KUKA KRL program: unicorn2_1.src

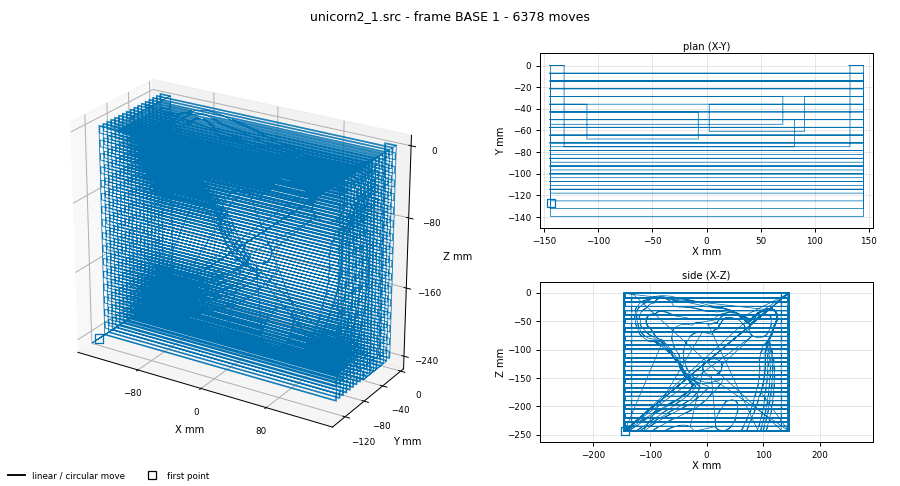
[picture p0: tool path of unicorn2_1.src in frame BASE 1, 6378 of 6379 moves have a stored position in this frame; points joined in program order, loops and branches not executed]
&ACCESS RVP
&REL 1
&PARAM TEMPLATE = C:\KRC\Roboter\Template\vorgabe
&PARAM EDITMASK = *
DEF unicorn2_1( )
EXT BAS (BAS_COMMAND :IN,REAL :IN )

INT INDX
FOR INDX=1 TO 6
	$ACC_AXIS[INDX]=50
	$VEL_AXIS[INDX]=20
ENDFOR

$VEL.ORI1=200
$VEL.ORI2=200
$ACC.ORI1=100
$ACC.ORI2=100

$VEL.CP = 0.2
$ACC.CP = 5

$IPO_MODE = #BASE
$APO.CDIS = 0.5
$ADVANCE = 5

$ACT_TOOL = 1
$TOOL=TOOL_DATA[1]
$ACT_BASE = 1
$BASE=BASE_DATA[1]

PTP {A1 30.0,A2 -90.0,A3 90.0,A4 0.0,A5 90.0,A6 0.0}

LIN {X -144.015,Y -126.800,Z -242.561,A -90.000,B 90.000,C 0.000} C_DIS
LIN {X -144.015,Y -114.300,Z -242.561,A -90.000,B 90.000,C 0.000} C_DIS
LIN {X 144.015,Y -114.300,Z -242.561,A -90.000,B 90.000,C 0.000} C_DIS
LIN {X 144.015,Y -114.300,Z -235.012,A -90.000,B 90.000,C 0.000} C_DIS
LIN {X -144.015,Y -114.300,Z -235.012,A -90.000,B 90.000,C 0.000} C_DIS
LIN {X -144.015,Y -114.300,Z -227.464,A -90.000,B 90.000,C 0.000} C_DIS
LIN {X 144.015,Y -114.300,Z -227.464,A -90.000,B 90.000,C 0.000} C_DIS
LIN {X 144.015,Y -114.300,Z -219.915,A -90.000,B 90.000,C 0.000} C_DIS
LIN {X -144.015,Y -114.300,Z -219.915,A -90.000,B 90.000,C 0.000} C_DIS
LIN {X -144.015,Y -114.300,Z -212.366,A -90.000,B 90.000,C 0.000} C_DIS
LIN {X 144.015,Y -114.300,Z -212.366,A -90.000,B 90.000,C 0.000} C_DIS
LIN {X 144.015,Y -114.300,Z -204.817,A -90.000,B 90.000,C 0.000} C_DIS
LIN {X -144.015,Y -114.300,Z -204.817,A -90.000,B 90.000,C 0.000} C_DIS
LIN {X -144.015,Y -114.300,Z -197.269,A -90.000,B 90.000,C 0.000} C_DIS
LIN {X 144.015,Y -114.300,Z -197.269,A -90.000,B 90.000,C 0.000} C_DIS
LIN {X 144.015,Y -114.300,Z -189.720,A -90.000,B 90.000,C 0.000} C_DIS
LIN {X -144.015,Y -114.300,Z -189.720,A -90.000,B 90.000,C 0.000} C_DIS
LIN {X -144.015,Y -114.300,Z -182.171,A -90.000,B 90.000,C 0.000} C_DIS
LIN {X 144.015,Y -114.300,Z -182.171,A -90.000,B 90.000,C 0.000} C_DIS
LIN {X 144.015,Y -114.300,Z -174.622,A -90.000,B 90.000,C 0.000} C_DIS
LIN {X -144.015,Y -114.300,Z -174.622,A -90.000,B 90.000,C 0.000} C_DIS
LIN {X -144.015,Y -114.300,Z -167.073,A -90.000,B 90.000,C 0.000} C_DIS
LIN {X 144.015,Y -114.300,Z -167.073,A -90.000,B 90.000,C 0.000} C_DIS
LIN {X 144.015,Y -114.300,Z -159.525,A -90.000,B 90.000,C 0.000} C_DIS
LIN {X -144.015,Y -114.300,Z -159.525,A -90.000,B 90.000,C 0.000} C_DIS
LIN {X -144.015,Y -114.300,Z -151.976,A -90.000,B 90.000,C 0.000} C_DIS
LIN {X 144.015,Y -114.300,Z -151.976,A -90.000,B 90.000,C 0.000} C_DIS
LIN {X 144.015,Y -114.300,Z -144.427,A -90.000,B 90.000,C 0.000} C_DIS
LIN {X -144.015,Y -114.300,Z -144.427,A -90.000,B 90.000,C 0.000} C_DIS
LIN {X -144.015,Y -114.300,Z -136.878,A -90.000,B 90.000,C 0.000} C_DIS
LIN {X 144.015,Y -114.300,Z -136.878,A -90.000,B 90.000,C 0.000} C_DIS
LIN {X 144.015,Y -114.300,Z -129.329,A -90.000,B 90.000,C 0.000} C_DIS
LIN {X -144.015,Y -114.300,Z -129.329,A -90.000,B 90.000,C 0.000} C_DIS
LIN {X -144.015,Y -114.300,Z -121.781,A -90.000,B 90.000,C 0.000} C_DIS
LIN {X 144.015,Y -114.300,Z -121.781,A -90.000,B 90.000,C 0.000} C_DIS
LIN {X 144.015,Y -114.300,Z -114.232,A -90.000,B 90.000,C 0.000} C_DIS
LIN {X -144.015,Y -114.300,Z -114.232,A -90.000,B 90.000,C 0.000} C_DIS
LIN {X -144.015,Y -114.300,Z -106.683,A -90.000,B 90.000,C 0.000} C_DIS
LIN {X 144.015,Y -114.300,Z -106.683,A -90.000,B 90.000,C 0.000} C_DIS
LIN {X 144.015,Y -114.300,Z -99.134,A -90.000,B 90.000,C 0.000} C_DIS
LIN {X -144.015,Y -114.300,Z -99.134,A -90.000,B 90.000,C 0.000} C_DIS
LIN {X -144.015,Y -114.300,Z -91.586,A -90.000,B 90.000,C 0.000} C_DIS
LIN {X 144.015,Y -114.300,Z -91.586,A -90.000,B 90.000,C 0.000} C_DIS
LIN {X 144.015,Y -114.300,Z -84.037,A -90.000,B 90.000,C 0.000} C_DIS
LIN {X -144.015,Y -114.300,Z -84.037,A -90.000,B 90.000,C 0.000} C_DIS
LIN {X -144.015,Y -114.300,Z -76.488,A -90.000,B 90.000,C 0.000} C_DIS
LIN {X 144.015,Y -114.300,Z -76.488,A -90.000,B 90.000,C 0.000} C_DIS
LIN {X 144.015,Y -114.300,Z -68.939,A -90.000,B 90.000,C 0.000} C_DIS
LIN {X -144.015,Y -114.300,Z -68.939,A -90.000,B 90.000,C 0.000} C_DIS
LIN {X -144.015,Y -114.300,Z -61.390,A -90.000,B 90.000,C 0.000} C_DIS
LIN {X 144.015,Y -114.300,Z -61.390,A -90.000,B 90.000,C 0.000} C_DIS
LIN {X 144.015,Y -114.300,Z -53.842,A -90.000,B 90.000,C 0.000} C_DIS
LIN {X -144.015,Y -114.300,Z -53.842,A -90.000,B 90.000,C 0.000} C_DIS
LIN {X -144.015,Y -114.300,Z -46.293,A -90.000,B 90.000,C 0.000} C_DIS
LIN {X 144.015,Y -114.300,Z -46.293,A -90.000,B 90.000,C 0.000} C_DIS
LIN {X 144.015,Y -114.300,Z -38.744,A -90.000,B 90.000,C 0.000} C_DIS
LIN {X -144.015,Y -114.300,Z -38.744,A -90.000,B 90.000,C 0.000} C_DIS
LIN {X -144.015,Y -114.300,Z -31.195,A -90.000,B 90.000,C 0.000} C_DIS
LIN {X 144.015,Y -114.300,Z -31.195,A -90.000,B 90.000,C 0.000} C_DIS
LIN {X 144.015,Y -114.300,Z -23.646,A -90.000,B 90.000,C 0.000} C_DIS
LIN {X -144.015,Y -114.300,Z -23.646,A -90.000,B 90.000,C 0.000} C_DIS
LIN {X -144.015,Y -114.300,Z -16.098,A -90.000,B 90.000,C 0.000} C_DIS
LIN {X 144.015,Y -114.300,Z -16.098,A -90.000,B 90.000,C 0.000} C_DIS
LIN {X 144.015,Y -114.300,Z -8.549,A -90.000,B 90.000,C 0.000} C_DIS
LIN {X -144.015,Y -114.300,Z -8.549,A -90.000,B 90.000,C 0.000} C_DIS
LIN {X -144.015,Y -114.300,Z -1.000,A -90.000,B 90.000,C 0.000} C_DIS
LIN {X 144.015,Y -114.300,Z -1.000,A -90.000,B 90.000,C 0.000} C_DIS
LIN {X 145.015,Y -114.300,Z 0.000,A -90.000,B 90.000,C 0.000} C_DIS
LIN {X -145.015,Y -114.300,Z 0.000,A -90.000,B 90.000,C 0.000} C_DIS
LIN {X -145.015,Y -114.300,Z -243.561,A -90.000,B 90.000,C 0.000} C_DIS
LIN {X 145.015,Y -114.300,Z -243.561,A -90.000,B 90.000,C 0.000} C_DIS
LIN {X 145.015,Y -114.300,Z 0.000,A -90.000,B 90.000,C 0.000} C_DIS
LIN {X 145.015,Y -126.800,Z 0.000,A -90.000,B 90.000,C 0.000} C_DIS
LIN {X 145.015,Y -139.300,Z 0.000,A -90.000,B 90.000,C 0.000} C_DIS
LIN {X -144.015,Y -139.300,Z -242.561,A -90.000,B 90.000,C 0.000} C_DIS
LIN {X -144.015,Y -132.156,Z -242.561,A -90.000,B 90.000,C 0.000} C_DIS
LIN {X -144.015,Y -119.656,Z -242.561,A -90.000,B 90.000,C 0.000} C_DIS
LIN {X -144.015,Y -107.156,Z -242.561,A -90.000,B 90.000,C 0.000} C_DIS
LIN {X 144.015,Y -107.156,Z -242.561,A -90.000,B 90.000,C 0.000} C_DIS
LIN {X 144.015,Y -107.156,Z -235.012,A -90.000,B 90.000,C 0.000} C_DIS
LIN {X -144.015,Y -107.156,Z -235.012,A -90.000,B 90.000,C 0.000} C_DIS
LIN {X -144.015,Y -107.156,Z -227.464,A -90.000,B 90.000,C 0.000} C_DIS
LIN {X 144.015,Y -107.156,Z -227.464,A -90.000,B 90.000,C 0.000} C_DIS
LIN {X 144.015,Y -107.156,Z -219.915,A -90.000,B 90.000,C 0.000} C_DIS
LIN {X -144.015,Y -107.156,Z -219.915,A -90.000,B 90.000,C 0.000} C_DIS
LIN {X -144.015,Y -107.156,Z -212.366,A -90.000,B 90.000,C 0.000} C_DIS
LIN {X 144.015,Y -107.156,Z -212.366,A -90.000,B 90.000,C 0.000} C_DIS
LIN {X 144.015,Y -107.156,Z -204.817,A -90.000,B 90.000,C 0.000} C_DIS
LIN {X -144.015,Y -107.156,Z -204.817,A -90.000,B 90.000,C 0.000} C_DIS
LIN {X -144.015,Y -107.156,Z -197.269,A -90.000,B 90.000,C 0.000} C_DIS
LIN {X 144.015,Y -107.156,Z -197.269,A -90.000,B 90.000,C 0.000} C_DIS
LIN {X 144.015,Y -107.156,Z -189.720,A -90.000,B 90.000,C 0.000} C_DIS
LIN {X -144.015,Y -107.156,Z -189.720,A -90.000,B 90.000,C 0.000} C_DIS
LIN {X -144.015,Y -107.156,Z -182.171,A -90.000,B 90.000,C 0.000} C_DIS
LIN {X 144.015,Y -107.156,Z -182.171,A -90.000,B 90.000,C 0.000} C_DIS
LIN {X 144.015,Y -107.156,Z -174.622,A -90.000,B 90.000,C 0.000} C_DIS
LIN {X -144.015,Y -107.156,Z -174.622,A -90.000,B 90.000,C 0.000} C_DIS
LIN {X -144.015,Y -107.156,Z -167.073,A -90.000,B 90.000,C 0.000} C_DIS
LIN {X 144.015,Y -107.156,Z -167.073,A -90.000,B 90.000,C 0.000} C_DIS
LIN {X 144.015,Y -107.156,Z -159.525,A -90.000,B 90.000,C 0.000} C_DIS
LIN {X -144.015,Y -107.156,Z -159.525,A -90.000,B 90.000,C 0.000} C_DIS
LIN {X -144.015,Y -107.156,Z -151.976,A -90.000,B 90.000,C 0.000} C_DIS
LIN {X 144.015,Y -107.156,Z -151.976,A -90.000,B 90.000,C 0.000} C_DIS
LIN {X 144.015,Y -107.156,Z -144.427,A -90.000,B 90.000,C 0.000} C_DIS
LIN {X -144.015,Y -107.156,Z -144.427,A -90.000,B 90.000,C 0.000} C_DIS
LIN {X -144.015,Y -107.156,Z -136.878,A -90.000,B 90.000,C 0.000} C_DIS
LIN {X 144.015,Y -107.156,Z -136.878,A -90.000,B 90.000,C 0.000} C_DIS
LIN {X 144.015,Y -107.156,Z -129.329,A -90.000,B 90.000,C 0.000} C_DIS
LIN {X -144.015,Y -107.156,Z -129.329,A -90.000,B 90.000,C 0.000} C_DIS
LIN {X -144.015,Y -107.156,Z -121.781,A -90.000,B 90.000,C 0.000} C_DIS
LIN {X 144.015,Y -107.156,Z -121.781,A -90.000,B 90.000,C 0.000} C_DIS
LIN {X 144.015,Y -107.156,Z -114.232,A -90.000,B 90.000,C 0.000} C_DIS
LIN {X -144.015,Y -107.156,Z -114.232,A -90.000,B 90.000,C 0.000} C_DIS
LIN {X -144.015,Y -107.156,Z -106.683,A -90.000,B 90.000,C 0.000} C_DIS
LIN {X 144.015,Y -107.156,Z -106.683,A -90.000,B 90.000,C 0.000} C_DIS
LIN {X 144.015,Y -107.156,Z -99.134,A -90.000,B 90.000,C 0.000} C_DIS
LIN {X -144.015,Y -107.156,Z -99.134,A -90.000,B 90.000,C 0.000} C_DIS
LIN {X -144.015,Y -107.156,Z -91.586,A -90.000,B 90.000,C 0.000} C_DIS
LIN {X 144.015,Y -107.156,Z -91.586,A -90.000,B 90.000,C 0.000} C_DIS
LIN {X 144.015,Y -107.156,Z -84.037,A -90.000,B 90.000,C 0.000} C_DIS
LIN {X -144.015,Y -107.156,Z -84.037,A -90.000,B 90.000,C 0.000} C_DIS
LIN {X -144.015,Y -107.156,Z -76.488,A -90.000,B 90.000,C 0.000} C_DIS
LIN {X 144.015,Y -107.156,Z -76.488,A -90.000,B 90.000,C 0.000} C_DIS
LIN {X 144.015,Y -107.156,Z -68.939,A -90.000,B 90.000,C 0.000} C_DIS
LIN {X -144.015,Y -107.156,Z -68.939,A -90.000,B 90.000,C 0.000} C_DIS
LIN {X -144.015,Y -107.156,Z -61.390,A -90.000,B 90.000,C 0.000} C_DIS
LIN {X 144.015,Y -107.156,Z -61.390,A -90.000,B 90.000,C 0.000} C_DIS
LIN {X 144.015,Y -107.156,Z -53.842,A -90.000,B 90.000,C 0.000} C_DIS
LIN {X -144.015,Y -107.156,Z -53.842,A -90.000,B 90.000,C 0.000} C_DIS
LIN {X -144.015,Y -107.156,Z -46.293,A -90.000,B 90.000,C 0.000} C_DIS
LIN {X 144.015,Y -107.156,Z -46.293,A -90.000,B 90.000,C 0.000} C_DIS
LIN {X 144.015,Y -107.156,Z -38.744,A -90.000,B 90.000,C 0.000} C_DIS
LIN {X -144.015,Y -107.156,Z -38.744,A -90.000,B 90.000,C 0.000} C_DIS
LIN {X -144.015,Y -107.156,Z -31.195,A -90.000,B 90.000,C 0.000} C_DIS
LIN {X 144.015,Y -107.156,Z -31.195,A -90.000,B 90.000,C 0.000} C_DIS
LIN {X 144.015,Y -107.156,Z -23.646,A -90.000,B 90.000,C 0.000} C_DIS
LIN {X -144.015,Y -107.156,Z -23.646,A -90.000,B 90.000,C 0.000} C_DIS
LIN {X -144.015,Y -107.156,Z -16.098,A -90.000,B 90.000,C 0.000} C_DIS
LIN {X 144.015,Y -107.156,Z -16.098,A -90.000,B 90.000,C 0.000} C_DIS
LIN {X 144.015,Y -107.156,Z -8.549,A -90.000,B 90.000,C 0.000} C_DIS
LIN {X -144.015,Y -107.156,Z -8.549,A -90.000,B 90.000,C 0.000} C_DIS
LIN {X -144.015,Y -107.156,Z -1.000,A -90.000,B 90.000,C 0.000} C_DIS
LIN {X 144.015,Y -107.156,Z -1.000,A -90.000,B 90.000,C 0.000} C_DIS
LIN {X 145.015,Y -107.156,Z 0.000,A -90.000,B 90.000,C 0.000} C_DIS
LIN {X -145.015,Y -107.156,Z 0.000,A -90.000,B 90.000,C 0.000} C_DIS
LIN {X -145.015,Y -107.156,Z -243.561,A -90.000,B 90.000,C 0.000} C_DIS
LIN {X 145.015,Y -107.156,Z -243.561,A -90.000,B 90.000,C 0.000} C_DIS
LIN {X 145.015,Y -107.156,Z 0.000,A -90.000,B 90.000,C 0.000} C_DIS
LIN {X 145.015,Y -119.656,Z 0.000,A -90.000,B 90.000,C 0.000} C_DIS
LIN {X 145.015,Y -132.156,Z 0.000,A -90.000,B 90.000,C 0.000} C_DIS
LIN {X -144.015,Y -132.156,Z -242.561,A -90.000,B 90.000,C 0.000} C_DIS
LIN {X -144.015,Y -125.013,Z -242.561,A -90.000,B 90.000,C 0.000} C_DIS
LIN {X -144.015,Y -112.513,Z -242.561,A -90.000,B 90.000,C 0.000} C_DIS
LIN {X -144.015,Y -100.013,Z -242.561,A -90.000,B 90.000,C 0.000} C_DIS
LIN {X 144.015,Y -100.013,Z -242.561,A -90.000,B 90.000,C 0.000} C_DIS
LIN {X 144.015,Y -100.013,Z -235.012,A -90.000,B 90.000,C 0.000} C_DIS
LIN {X -144.015,Y -100.013,Z -235.012,A -90.000,B 90.000,C 0.000} C_DIS
LIN {X -144.015,Y -100.013,Z -227.464,A -90.000,B 90.000,C 0.000} C_DIS
LIN {X 144.015,Y -100.013,Z -227.464,A -90.000,B 90.000,C 0.000} C_DIS
LIN {X 144.015,Y -100.013,Z -219.915,A -90.000,B 90.000,C 0.000} C_DIS
LIN {X -144.015,Y -100.013,Z -219.915,A -90.000,B 90.000,C 0.000} C_DIS
LIN {X -144.015,Y -100.013,Z -212.366,A -90.000,B 90.000,C 0.000} C_DIS
LIN {X 144.015,Y -100.013,Z -212.366,A -90.000,B 90.000,C 0.000} C_DIS
LIN {X 144.015,Y -100.013,Z -204.817,A -90.000,B 90.000,C 0.000} C_DIS
LIN {X -144.015,Y -100.013,Z -204.817,A -90.000,B 90.000,C 0.000} C_DIS
LIN {X -144.015,Y -100.013,Z -197.269,A -90.000,B 90.000,C 0.000} C_DIS
LIN {X 144.015,Y -100.013,Z -197.269,A -90.000,B 90.000,C 0.000} C_DIS
LIN {X 144.015,Y -100.013,Z -189.720,A -90.000,B 90.000,C 0.000} C_DIS
LIN {X -144.015,Y -100.013,Z -189.720,A -90.000,B 90.000,C 0.000} C_DIS
LIN {X -144.015,Y -100.013,Z -182.171,A -90.000,B 90.000,C 0.000} C_DIS
LIN {X 144.015,Y -100.013,Z -182.171,A -90.000,B 90.000,C 0.000} C_DIS
LIN {X 144.015,Y -100.013,Z -174.622,A -90.000,B 90.000,C 0.000} C_DIS
LIN {X -144.015,Y -100.013,Z -174.622,A -90.000,B 90.000,C 0.000} C_DIS
LIN {X -144.015,Y -100.013,Z -167.073,A -90.000,B 90.000,C 0.000} C_DIS
LIN {X 144.015,Y -100.013,Z -167.073,A -90.000,B 90.000,C 0.000} C_DIS
LIN {X 144.015,Y -100.013,Z -159.525,A -90.000,B 90.000,C 0.000} C_DIS
LIN {X -144.015,Y -100.013,Z -159.525,A -90.000,B 90.000,C 0.000} C_DIS
LIN {X -144.015,Y -100.013,Z -151.976,A -90.000,B 90.000,C 0.000} C_DIS
LIN {X 144.015,Y -100.013,Z -151.976,A -90.000,B 90.000,C 0.000} C_DIS
LIN {X 144.015,Y -100.013,Z -144.427,A -90.000,B 90.000,C 0.000} C_DIS
LIN {X -144.015,Y -100.013,Z -144.427,A -90.000,B 90.000,C 0.000} C_DIS
LIN {X -144.015,Y -100.013,Z -136.878,A -90.000,B 90.000,C 0.000} C_DIS
LIN {X 144.015,Y -100.013,Z -136.878,A -90.000,B 90.000,C 0.000} C_DIS
LIN {X 144.015,Y -100.013,Z -129.329,A -90.000,B 90.000,C 0.000} C_DIS
LIN {X -144.015,Y -100.013,Z -129.329,A -90.000,B 90.000,C 0.000} C_DIS
LIN {X -144.015,Y -100.013,Z -121.781,A -90.000,B 90.000,C 0.000} C_DIS
LIN {X 144.015,Y -100.013,Z -121.781,A -90.000,B 90.000,C 0.000} C_DIS
LIN {X 144.015,Y -100.013,Z -114.232,A -90.000,B 90.000,C 0.000} C_DIS
LIN {X -144.015,Y -100.013,Z -114.232,A -90.000,B 90.000,C 0.000} C_DIS
LIN {X -144.015,Y -100.013,Z -106.683,A -90.000,B 90.000,C 0.000} C_DIS
LIN {X 144.015,Y -100.013,Z -106.683,A -90.000,B 90.000,C 0.000} C_DIS
LIN {X 144.015,Y -100.013,Z -99.134,A -90.000,B 90.000,C 0.000} C_DIS
LIN {X -144.015,Y -100.013,Z -99.134,A -90.000,B 90.000,C 0.000} C_DIS
LIN {X -144.015,Y -100.013,Z -91.586,A -90.000,B 90.000,C 0.000} C_DIS
LIN {X 144.015,Y -100.013,Z -91.586,A -90.000,B 90.000,C 0.000} C_DIS
LIN {X 144.015,Y -100.013,Z -84.037,A -90.000,B 90.000,C 0.000} C_DIS
LIN {X -144.015,Y -100.013,Z -84.037,A -90.000,B 90.000,C 0.000} C_DIS
LIN {X -144.015,Y -100.013,Z -76.488,A -90.000,B 90.000,C 0.000} C_DIS
LIN {X 144.015,Y -100.013,Z -76.488,A -90.000,B 90.000,C 0.000} C_DIS
LIN {X 144.015,Y -100.013,Z -68.939,A -90.000,B 90.000,C 0.000} C_DIS
LIN {X -144.015,Y -100.013,Z -68.939,A -90.000,B 90.000,C 0.000} C_DIS
LIN {X -144.015,Y -100.013,Z -61.390,A -90.000,B 90.000,C 0.000} C_DIS
LIN {X 144.015,Y -100.013,Z -61.390,A -90.000,B 90.000,C 0.000} C_DIS
LIN {X 144.015,Y -100.013,Z -53.842,A -90.000,B 90.000,C 0.000} C_DIS
LIN {X -144.015,Y -100.013,Z -53.842,A -90.000,B 90.000,C 0.000} C_DIS
LIN {X -144.015,Y -100.013,Z -46.293,A -90.000,B 90.000,C 0.000} C_DIS
LIN {X 144.015,Y -100.013,Z -46.293,A -90.000,B 90.000,C 0.000} C_DIS
LIN {X 144.015,Y -100.013,Z -38.744,A -90.000,B 90.000,C 0.000} C_DIS
LIN {X -144.015,Y -100.013,Z -38.744,A -90.000,B 90.000,C 0.000} C_DIS
LIN {X -144.015,Y -100.013,Z -31.195,A -90.000,B 90.000,C 0.000} C_DIS
LIN {X 144.015,Y -100.013,Z -31.195,A -90.000,B 90.000,C 0.000} C_DIS
LIN {X 144.015,Y -100.013,Z -23.646,A -90.000,B 90.000,C 0.000} C_DIS
LIN {X -144.015,Y -100.013,Z -23.646,A -90.000,B 90.000,C 0.000} C_DIS
LIN {X -144.015,Y -100.013,Z -16.098,A -90.000,B 90.000,C 0.000} C_DIS
LIN {X 144.015,Y -100.013,Z -16.098,A -90.000,B 90.000,C 0.000} C_DIS
LIN {X 144.015,Y -100.013,Z -8.549,A -90.000,B 90.000,C 0.000} C_DIS
LIN {X -144.015,Y -100.013,Z -8.549,A -90.000,B 90.000,C 0.000} C_DIS
LIN {X -144.015,Y -100.013,Z -1.000,A -90.000,B 90.000,C 0.000} C_DIS
LIN {X 144.015,Y -100.013,Z -1.000,A -90.000,B 90.000,C 0.000} C_DIS
LIN {X 145.015,Y -100.013,Z 0.000,A -90.000,B 90.000,C 0.000} C_DIS
LIN {X -145.015,Y -100.013,Z 0.000,A -90.000,B 90.000,C 0.000} C_DIS
LIN {X -145.015,Y -100.013,Z -243.561,A -90.000,B 90.000,C 0.000} C_DIS
LIN {X 145.015,Y -100.013,Z -243.561,A -90.000,B 90.000,C 0.000} C_DIS
LIN {X 145.015,Y -100.013,Z 0.000,A -90.000,B 90.000,C 0.000} C_DIS
LIN {X 145.015,Y -112.513,Z 0.000,A -90.000,B 90.000,C 0.000} C_DIS
LIN {X 145.015,Y -125.013,Z 0.000,A -90.000,B 90.000,C 0.000} C_DIS
LIN {X -144.015,Y -125.013,Z -242.561,A -90.000,B 90.000,C 0.000} C_DIS
LIN {X -144.015,Y -117.869,Z -242.561,A -90.000,B 90.000,C 0.000} C_DIS
LIN {X -144.015,Y -105.369,Z -242.561,A -90.000,B 90.000,C 0.000} C_DIS
LIN {X -144.015,Y -92.869,Z -242.561,A -90.000,B 90.000,C 0.000} C_DIS
LIN {X 144.015,Y -92.869,Z -242.561,A -90.000,B 90.000,C 0.000} C_DIS
LIN {X 144.015,Y -92.869,Z -235.012,A -90.000,B 90.000,C 0.000} C_DIS
LIN {X -144.015,Y -92.869,Z -235.012,A -90.000,B 90.000,C 0.000} C_DIS
LIN {X -144.015,Y -92.869,Z -227.464,A -90.000,B 90.000,C 0.000} C_DIS
LIN {X 144.015,Y -92.869,Z -227.464,A -90.000,B 90.000,C 0.000} C_DIS
LIN {X 144.015,Y -92.869,Z -219.915,A -90.000,B 90.000,C 0.000} C_DIS
LIN {X -144.015,Y -92.869,Z -219.915,A -90.000,B 90.000,C 0.000} C_DIS
LIN {X -144.015,Y -92.869,Z -212.366,A -90.000,B 90.000,C 0.000} C_DIS
LIN {X 144.015,Y -92.869,Z -212.366,A -90.000,B 90.000,C 0.000} C_DIS
LIN {X 144.015,Y -92.869,Z -204.817,A -90.000,B 90.000,C 0.000} C_DIS
LIN {X -144.015,Y -92.869,Z -204.817,A -90.000,B 90.000,C 0.000} C_DIS
LIN {X -144.015,Y -92.869,Z -197.269,A -90.000,B 90.000,C 0.000} C_DIS
LIN {X 144.015,Y -92.869,Z -197.269,A -90.000,B 90.000,C 0.000} C_DIS
LIN {X 144.015,Y -92.869,Z -189.720,A -90.000,B 90.000,C 0.000} C_DIS
LIN {X -144.015,Y -92.869,Z -189.720,A -90.000,B 90.000,C 0.000} C_DIS
LIN {X -144.015,Y -92.869,Z -182.171,A -90.000,B 90.000,C 0.000} C_DIS
LIN {X 144.015,Y -92.869,Z -182.171,A -90.000,B 90.000,C 0.000} C_DIS
LIN {X 144.015,Y -92.869,Z -174.622,A -90.000,B 90.000,C 0.000} C_DIS
LIN {X -144.015,Y -92.869,Z -174.622,A -90.000,B 90.000,C 0.000} C_DIS
LIN {X -144.015,Y -92.869,Z -167.073,A -90.000,B 90.000,C 0.000} C_DIS
LIN {X 144.015,Y -92.869,Z -167.073,A -90.000,B 90.000,C 0.000} C_DIS
LIN {X 144.015,Y -92.869,Z -159.525,A -90.000,B 90.000,C 0.000} C_DIS
LIN {X -144.015,Y -92.869,Z -159.525,A -90.000,B 90.000,C 0.000} C_DIS
LIN {X -144.015,Y -92.869,Z -151.976,A -90.000,B 90.000,C 0.000} C_DIS
LIN {X 144.015,Y -92.869,Z -151.976,A -90.000,B 90.000,C 0.000} C_DIS
LIN {X 144.015,Y -92.869,Z -144.427,A -90.000,B 90.000,C 0.000} C_DIS
LIN {X -144.015,Y -92.869,Z -144.427,A -90.000,B 90.000,C 0.000} C_DIS
LIN {X -144.015,Y -92.869,Z -136.878,A -90.000,B 90.000,C 0.000} C_DIS
LIN {X 144.015,Y -92.869,Z -136.878,A -90.000,B 90.000,C 0.000} C_DIS
LIN {X 144.015,Y -92.869,Z -129.329,A -90.000,B 90.000,C 0.000} C_DIS
LIN {X -144.015,Y -92.869,Z -129.329,A -90.000,B 90.000,C 0.000} C_DIS
LIN {X -144.015,Y -92.869,Z -121.781,A -90.000,B 90.000,C 0.000} C_DIS
LIN {X 144.015,Y -92.869,Z -121.781,A -90.000,B 90.000,C 0.000} C_DIS
LIN {X 144.015,Y -92.869,Z -114.232,A -90.000,B 90.000,C 0.000} C_DIS
LIN {X -144.015,Y -92.869,Z -114.232,A -90.000,B 90.000,C 0.000} C_DIS
LIN {X -144.015,Y -92.869,Z -106.683,A -90.000,B 90.000,C 0.000} C_DIS
LIN {X 144.015,Y -92.869,Z -106.683,A -90.000,B 90.000,C 0.000} C_DIS
LIN {X 144.015,Y -92.869,Z -99.134,A -90.000,B 90.000,C 0.000} C_DIS
LIN {X -144.015,Y -92.869,Z -99.134,A -90.000,B 90.000,C 0.000} C_DIS
LIN {X -144.015,Y -92.869,Z -91.586,A -90.000,B 90.000,C 0.000} C_DIS
LIN {X 144.015,Y -92.869,Z -91.586,A -90.000,B 90.000,C 0.000} C_DIS
LIN {X 144.015,Y -92.869,Z -84.037,A -90.000,B 90.000,C 0.000} C_DIS
LIN {X -144.015,Y -92.869,Z -84.037,A -90.000,B 90.000,C 0.000} C_DIS
LIN {X -144.015,Y -92.869,Z -76.488,A -90.000,B 90.000,C 0.000} C_DIS
LIN {X 144.015,Y -92.869,Z -76.488,A -90.000,B 90.000,C 0.000} C_DIS
LIN {X 144.015,Y -92.869,Z -68.939,A -90.000,B 90.000,C 0.000} C_DIS
LIN {X -144.015,Y -92.869,Z -68.939,A -90.000,B 90.000,C 0.000} C_DIS
LIN {X -144.015,Y -92.869,Z -61.390,A -90.000,B 90.000,C 0.000} C_DIS
LIN {X 144.015,Y -92.869,Z -61.390,A -90.000,B 90.000,C 0.000} C_DIS
LIN {X 144.015,Y -92.869,Z -53.842,A -90.000,B 90.000,C 0.000} C_DIS
LIN {X -144.015,Y -92.869,Z -53.842,A -90.000,B 90.000,C 0.000} C_DIS
LIN {X -144.015,Y -92.869,Z -46.293,A -90.000,B 90.000,C 0.000} C_DIS
LIN {X 144.015,Y -92.869,Z -46.293,A -90.000,B 90.000,C 0.000} C_DIS
LIN {X 144.015,Y -92.869,Z -38.744,A -90.000,B 90.000,C 0.000} C_DIS
LIN {X -144.015,Y -92.869,Z -38.744,A -90.000,B 90.000,C 0.000} C_DIS
LIN {X -144.015,Y -92.869,Z -31.195,A -90.000,B 90.000,C 0.000} C_DIS
LIN {X 144.015,Y -92.869,Z -31.195,A -90.000,B 90.000,C 0.000} C_DIS
LIN {X 144.015,Y -92.869,Z -23.646,A -90.000,B 90.000,C 0.000} C_DIS
LIN {X -144.015,Y -92.869,Z -23.646,A -90.000,B 90.000,C 0.000} C_DIS
LIN {X -144.015,Y -92.869,Z -16.098,A -90.000,B 90.000,C 0.000} C_DIS
LIN {X 144.015,Y -92.869,Z -16.098,A -90.000,B 90.000,C 0.000} C_DIS
LIN {X 144.015,Y -92.869,Z -8.549,A -90.000,B 90.000,C 0.000} C_DIS
LIN {X -144.015,Y -92.869,Z -8.549,A -90.000,B 90.000,C 0.000} C_DIS
LIN {X -144.015,Y -92.869,Z -1.000,A -90.000,B 90.000,C 0.000} C_DIS
LIN {X 144.015,Y -92.869,Z -1.000,A -90.000,B 90.000,C 0.000} C_DIS
LIN {X 145.015,Y -92.869,Z 0.000,A -90.000,B 90.000,C 0.000} C_DIS
LIN {X -145.015,Y -92.869,Z 0.000,A -90.000,B 90.000,C 0.000} C_DIS
LIN {X -145.015,Y -92.869,Z -243.561,A -90.000,B 90.000,C 0.000} C_DIS
LIN {X 145.015,Y -92.869,Z -243.561,A -90.000,B 90.000,C 0.000} C_DIS
LIN {X 145.015,Y -92.869,Z 0.000,A -90.000,B 90.000,C 0.000} C_DIS
LIN {X 145.015,Y -105.369,Z 0.000,A -90.000,B 90.000,C 0.000} C_DIS
LIN {X 145.015,Y -117.869,Z 0.000,A -90.000,B 90.000,C 0.000} C_DIS
LIN {X -144.015,Y -117.869,Z -242.561,A -90.000,B 90.000,C 0.000} C_DIS
LIN {X -144.015,Y -110.725,Z -242.561,A -90.000,B 90.000,C 0.000} C_DIS
LIN {X -144.015,Y -98.225,Z -242.561,A -90.000,B 90.000,C 0.000} C_DIS
LIN {X -144.015,Y -85.725,Z -242.561,A -90.000,B 90.000,C 0.000} C_DIS
LIN {X 144.015,Y -85.725,Z -242.561,A -90.000,B 90.000,C 0.000} C_DIS
LIN {X 144.015,Y -85.725,Z -235.012,A -90.000,B 90.000,C 0.000} C_DIS
LIN {X -144.015,Y -85.725,Z -235.012,A -90.000,B 90.000,C 0.000} C_DIS
LIN {X -144.015,Y -85.725,Z -227.464,A -90.000,B 90.000,C 0.000} C_DIS
LIN {X 144.015,Y -85.725,Z -227.464,A -90.000,B 90.000,C 0.000} C_DIS
LIN {X 144.015,Y -85.725,Z -219.915,A -90.000,B 90.000,C 0.000} C_DIS
LIN {X -144.015,Y -85.725,Z -219.915,A -90.000,B 90.000,C 0.000} C_DIS
LIN {X -144.015,Y -85.725,Z -212.366,A -90.000,B 90.000,C 0.000} C_DIS
LIN {X 144.015,Y -85.725,Z -212.366,A -90.000,B 90.000,C 0.000} C_DIS
LIN {X 144.015,Y -85.725,Z -204.817,A -90.000,B 90.000,C 0.000} C_DIS
LIN {X -144.015,Y -85.725,Z -204.817,A -90.000,B 90.000,C 0.000} C_DIS
LIN {X -144.015,Y -85.725,Z -197.269,A -90.000,B 90.000,C 0.000} C_DIS
LIN {X 144.015,Y -85.725,Z -197.269,A -90.000,B 90.000,C 0.000} C_DIS
LIN {X 144.015,Y -85.725,Z -189.720,A -90.000,B 90.000,C 0.000} C_DIS
LIN {X -144.015,Y -85.725,Z -189.720,A -90.000,B 90.000,C 0.000} C_DIS
LIN {X -144.015,Y -85.725,Z -182.171,A -90.000,B 90.000,C 0.000} C_DIS
LIN {X 144.015,Y -85.725,Z -182.171,A -90.000,B 90.000,C 0.000} C_DIS
LIN {X 144.015,Y -85.725,Z -174.622,A -90.000,B 90.000,C 0.000} C_DIS
LIN {X -144.015,Y -85.725,Z -174.622,A -90.000,B 90.000,C 0.000} C_DIS
LIN {X -144.015,Y -85.725,Z -167.073,A -90.000,B 90.000,C 0.000} C_DIS
LIN {X 144.015,Y -85.725,Z -167.073,A -90.000,B 90.000,C 0.000} C_DIS
LIN {X 144.015,Y -85.725,Z -159.525,A -90.000,B 90.000,C 0.000} C_DIS
LIN {X -144.015,Y -85.725,Z -159.525,A -90.000,B 90.000,C 0.000} C_DIS
LIN {X -144.015,Y -85.725,Z -151.976,A -90.000,B 90.000,C 0.000} C_DIS
LIN {X 144.015,Y -85.725,Z -151.976,A -90.000,B 90.000,C 0.000} C_DIS
LIN {X 144.015,Y -85.725,Z -144.427,A -90.000,B 90.000,C 0.000} C_DIS
LIN {X -144.015,Y -85.725,Z -144.427,A -90.000,B 90.000,C 0.000} C_DIS
LIN {X -144.015,Y -85.725,Z -136.878,A -90.000,B 90.000,C 0.000} C_DIS
LIN {X 144.015,Y -85.725,Z -136.878,A -90.000,B 90.000,C 0.000} C_DIS
LIN {X 144.015,Y -85.725,Z -129.329,A -90.000,B 90.000,C 0.000} C_DIS
LIN {X -144.015,Y -85.725,Z -129.329,A -90.000,B 90.000,C 0.000} C_DIS
LIN {X -144.015,Y -85.725,Z -121.781,A -90.000,B 90.000,C 0.000} C_DIS
LIN {X 144.015,Y -85.725,Z -121.781,A -90.000,B 90.000,C 0.000} C_DIS
LIN {X 144.015,Y -85.725,Z -114.232,A -90.000,B 90.000,C 0.000} C_DIS
LIN {X -144.015,Y -85.725,Z -114.232,A -90.000,B 90.000,C 0.000} C_DIS
LIN {X -144.015,Y -85.725,Z -106.683,A -90.000,B 90.000,C 0.000} C_DIS
LIN {X 144.015,Y -85.725,Z -106.683,A -90.000,B 90.000,C 0.000} C_DIS
LIN {X 144.015,Y -85.725,Z -99.134,A -90.000,B 90.000,C 0.000} C_DIS
LIN {X -144.015,Y -85.725,Z -99.134,A -90.000,B 90.000,C 0.000} C_DIS
LIN {X -144.015,Y -85.725,Z -91.586,A -90.000,B 90.000,C 0.000} C_DIS
LIN {X 144.015,Y -85.725,Z -91.586,A -90.000,B 90.000,C 0.000} C_DIS
LIN {X 144.015,Y -85.725,Z -84.037,A -90.000,B 90.000,C 0.000} C_DIS
LIN {X -144.015,Y -85.725,Z -84.037,A -90.000,B 90.000,C 0.000} C_DIS
LIN {X -144.015,Y -85.725,Z -76.488,A -90.000,B 90.000,C 0.000} C_DIS
LIN {X 144.015,Y -85.725,Z -76.488,A -90.000,B 90.000,C 0.000} C_DIS
LIN {X 144.015,Y -85.725,Z -68.939,A -90.000,B 90.000,C 0.000} C_DIS
LIN {X -144.015,Y -85.725,Z -68.939,A -90.000,B 90.000,C 0.000} C_DIS
LIN {X -144.015,Y -85.725,Z -61.390,A -90.000,B 90.000,C 0.000} C_DIS
LIN {X 144.015,Y -85.725,Z -61.390,A -90.000,B 90.000,C 0.000} C_DIS
LIN {X 144.015,Y -85.725,Z -53.842,A -90.000,B 90.000,C 0.000} C_DIS
LIN {X -144.015,Y -85.725,Z -53.842,A -90.000,B 90.000,C 0.000} C_DIS
LIN {X -144.015,Y -85.725,Z -46.293,A -90.000,B 90.000,C 0.000} C_DIS
LIN {X 144.015,Y -85.725,Z -46.293,A -90.000,B 90.000,C 0.000} C_DIS
LIN {X 144.015,Y -85.725,Z -38.744,A -90.000,B 90.000,C 0.000} C_DIS
LIN {X -144.015,Y -85.725,Z -38.744,A -90.000,B 90.000,C 0.000} C_DIS
LIN {X -144.015,Y -85.725,Z -31.195,A -90.000,B 90.000,C 0.000} C_DIS
LIN {X 144.015,Y -85.725,Z -31.195,A -90.000,B 90.000,C 0.000} C_DIS
LIN {X 144.015,Y -85.725,Z -23.646,A -90.000,B 90.000,C 0.000} C_DIS
LIN {X -144.015,Y -85.725,Z -23.646,A -90.000,B 90.000,C 0.000} C_DIS
LIN {X -144.015,Y -85.725,Z -16.098,A -90.000,B 90.000,C 0.000} C_DIS
LIN {X 144.015,Y -85.725,Z -16.098,A -90.000,B 90.000,C 0.000} C_DIS
LIN {X 144.015,Y -85.725,Z -8.549,A -90.000,B 90.000,C 0.000} C_DIS
LIN {X -144.015,Y -85.725,Z -8.549,A -90.000,B 90.000,C 0.000} C_DIS
LIN {X -144.015,Y -85.725,Z -1.000,A -90.000,B 90.000,C 0.000} C_DIS
LIN {X 144.015,Y -85.725,Z -1.000,A -90.000,B 90.000,C 0.000} C_DIS
LIN {X 145.015,Y -85.725,Z 0.000,A -90.000,B 90.000,C 0.000} C_DIS
LIN {X -145.015,Y -85.725,Z 0.000,A -90.000,B 90.000,C 0.000} C_DIS
LIN {X -145.015,Y -85.725,Z -243.561,A -90.000,B 90.000,C 0.000} C_DIS
LIN {X 145.015,Y -85.725,Z -243.561,A -90.000,B 90.000,C 0.000} C_DIS
LIN {X 145.015,Y -85.725,Z 0.000,A -90.000,B 90.000,C 0.000} C_DIS
LIN {X 145.015,Y -98.225,Z 0.000,A -90.000,B 90.000,C 0.000} C_DIS
LIN {X 145.015,Y -110.725,Z 0.000,A -90.000,B 90.000,C 0.000} C_DIS
LIN {X -144.015,Y -110.725,Z -242.561,A -90.000,B 90.000,C 0.000} C_DIS
LIN {X -144.015,Y -103.581,Z -242.561,A -90.000,B 90.000,C 0.000} C_DIS
LIN {X -144.015,Y -91.081,Z -242.561,A -90.000,B 90.000,C 0.000} C_DIS
LIN {X -144.015,Y -78.581,Z -242.561,A -90.000,B 90.000,C 0.000} C_DIS
LIN {X 144.015,Y -78.581,Z -242.561,A -90.000,B 90.000,C 0.000} C_DIS
LIN {X 144.015,Y -78.581,Z -235.012,A -90.000,B 90.000,C 0.000} C_DIS
LIN {X -144.015,Y -78.581,Z -235.012,A -90.000,B 90.000,C 0.000} C_DIS
LIN {X -144.015,Y -78.581,Z -227.464,A -90.000,B 90.000,C 0.000} C_DIS
LIN {X 144.015,Y -78.581,Z -227.464,A -90.000,B 90.000,C 0.000} C_DIS
LIN {X 144.015,Y -78.581,Z -219.915,A -90.000,B 90.000,C 0.000} C_DIS
LIN {X -144.015,Y -78.581,Z -219.915,A -90.000,B 90.000,C 0.000} C_DIS
LIN {X -144.015,Y -78.581,Z -212.366,A -90.000,B 90.000,C 0.000} C_DIS
LIN {X 144.015,Y -78.581,Z -212.366,A -90.000,B 90.000,C 0.000} C_DIS
LIN {X 144.015,Y -78.581,Z -204.817,A -90.000,B 90.000,C 0.000} C_DIS
LIN {X -144.015,Y -78.581,Z -204.817,A -90.000,B 90.000,C 0.000} C_DIS
LIN {X -144.015,Y -78.581,Z -197.269,A -90.000,B 90.000,C 0.000} C_DIS
LIN {X 144.015,Y -78.581,Z -197.269,A -90.000,B 90.000,C 0.000} C_DIS
LIN {X 144.015,Y -78.581,Z -189.720,A -90.000,B 90.000,C 0.000} C_DIS
LIN {X -144.015,Y -78.581,Z -189.720,A -90.000,B 90.000,C 0.000} C_DIS
LIN {X -144.015,Y -78.581,Z -182.171,A -90.000,B 90.000,C 0.000} C_DIS
LIN {X 144.015,Y -78.581,Z -182.171,A -90.000,B 90.000,C 0.000} C_DIS
LIN {X 144.015,Y -78.581,Z -174.622,A -90.000,B 90.000,C 0.000} C_DIS
LIN {X -144.015,Y -78.581,Z -174.622,A -90.000,B 90.000,C 0.000} C_DIS
LIN {X -144.015,Y -78.581,Z -167.073,A -90.000,B 90.000,C 0.000} C_DIS
LIN {X 144.015,Y -78.581,Z -167.073,A -90.000,B 90.000,C 0.000} C_DIS
LIN {X 144.015,Y -78.581,Z -159.525,A -90.000,B 90.000,C 0.000} C_DIS
LIN {X -144.015,Y -78.581,Z -159.525,A -90.000,B 90.000,C 0.000} C_DIS
LIN {X -144.015,Y -78.581,Z -151.976,A -90.000,B 90.000,C 0.000} C_DIS
LIN {X 144.015,Y -78.581,Z -151.976,A -90.000,B 90.000,C 0.000} C_DIS
LIN {X 144.015,Y -78.581,Z -144.427,A -90.000,B 90.000,C 0.000} C_DIS
LIN {X -144.015,Y -78.581,Z -144.427,A -90.000,B 90.000,C 0.000} C_DIS
LIN {X -144.015,Y -78.581,Z -136.878,A -90.000,B 90.000,C 0.000} C_DIS
LIN {X 144.015,Y -78.581,Z -136.878,A -90.000,B 90.000,C 0.000} C_DIS
LIN {X 144.015,Y -78.581,Z -129.329,A -90.000,B 90.000,C 0.000} C_DIS
LIN {X -144.015,Y -78.581,Z -129.329,A -90.000,B 90.000,C 0.000} C_DIS
LIN {X -144.015,Y -78.581,Z -121.781,A -90.000,B 90.000,C 0.000} C_DIS
LIN {X 144.015,Y -78.581,Z -121.781,A -90.000,B 90.000,C 0.000} C_DIS
LIN {X 144.015,Y -78.581,Z -114.232,A -90.000,B 90.000,C 0.000} C_DIS
LIN {X -144.015,Y -78.581,Z -114.232,A -90.000,B 90.000,C 0.000} C_DIS
LIN {X -144.015,Y -78.581,Z -106.683,A -90.000,B 90.000,C 0.000} C_DIS
LIN {X 144.015,Y -78.581,Z -106.683,A -90.000,B 90.000,C 0.000} C_DIS
LIN {X 144.015,Y -78.581,Z -99.134,A -90.000,B 90.000,C 0.000} C_DIS
LIN {X -144.015,Y -78.581,Z -99.134,A -90.000,B 90.000,C 0.000} C_DIS
LIN {X -144.015,Y -78.581,Z -91.586,A -90.000,B 90.000,C 0.000} C_DIS
LIN {X 144.015,Y -78.581,Z -91.586,A -90.000,B 90.000,C 0.000} C_DIS
LIN {X 144.015,Y -78.581,Z -84.037,A -90.000,B 90.000,C 0.000} C_DIS
LIN {X -144.015,Y -78.581,Z -84.037,A -90.000,B 90.000,C 0.000} C_DIS
LIN {X -144.015,Y -78.581,Z -76.488,A -90.000,B 90.000,C 0.000} C_DIS
LIN {X 144.015,Y -78.581,Z -76.488,A -90.000,B 90.000,C 0.000} C_DIS
LIN {X 144.015,Y -78.581,Z -68.939,A -90.000,B 90.000,C 0.000} C_DIS
LIN {X -144.015,Y -78.581,Z -68.939,A -90.000,B 90.000,C 0.000} C_DIS
LIN {X -144.015,Y -78.581,Z -61.390,A -90.000,B 90.000,C 0.000} C_DIS
LIN {X 144.015,Y -78.581,Z -61.390,A -90.000,B 90.000,C 0.000} C_DIS
LIN {X 144.015,Y -78.581,Z -53.842,A -90.000,B 90.000,C 0.000} C_DIS
LIN {X -144.015,Y -78.581,Z -53.842,A -90.000,B 90.000,C 0.000} C_DIS
LIN {X -144.015,Y -78.581,Z -46.293,A -90.000,B 90.000,C 0.000} C_DIS
LIN {X 144.015,Y -78.581,Z -46.293,A -90.000,B 90.000,C 0.000} C_DIS
LIN {X 144.015,Y -78.581,Z -38.744,A -90.000,B 90.000,C 0.000} C_DIS
LIN {X -144.015,Y -78.581,Z -38.744,A -90.000,B 90.000,C 0.000} C_DIS
LIN {X -144.015,Y -78.581,Z -31.195,A -90.000,B 90.000,C 0.000} C_DIS
LIN {X 144.015,Y -78.581,Z -31.195,A -90.000,B 90.000,C 0.000} C_DIS
LIN {X 144.015,Y -78.581,Z -23.646,A -90.000,B 90.000,C 0.000} C_DIS
LIN {X -144.015,Y -78.581,Z -23.646,A -90.000,B 90.000,C 0.000} C_DIS
LIN {X -144.015,Y -78.581,Z -16.098,A -90.000,B 90.000,C 0.000} C_DIS
LIN {X 144.015,Y -78.581,Z -16.098,A -90.000,B 90.000,C 0.000} C_DIS
LIN {X 144.015,Y -78.581,Z -8.549,A -90.000,B 90.000,C 0.000} C_DIS
LIN {X -144.015,Y -78.581,Z -8.549,A -90.000,B 90.000,C 0.000} C_DIS
LIN {X -144.015,Y -78.581,Z -1.000,A -90.000,B 90.000,C 0.000} C_DIS
LIN {X 144.015,Y -78.581,Z -1.000,A -90.000,B 90.000,C 0.000} C_DIS
LIN {X 145.015,Y -78.581,Z 0.000,A -90.000,B 90.000,C 0.000} C_DIS
LIN {X -145.015,Y -78.581,Z 0.000,A -90.000,B 90.000,C 0.000} C_DIS
LIN {X -145.015,Y -78.581,Z -243.561,A -90.000,B 90.000,C 0.000} C_DIS
LIN {X 145.015,Y -78.581,Z -243.561,A -90.000,B 90.000,C 0.000} C_DIS
LIN {X 145.015,Y -78.581,Z 0.000,A -90.000,B 90.000,C 0.000} C_DIS
LIN {X 145.015,Y -91.081,Z 0.000,A -90.000,B 90.000,C 0.000} C_DIS
LIN {X 145.015,Y -103.581,Z 0.000,A -90.000,B 90.000,C 0.000} C_DIS
LIN {X -144.015,Y -103.581,Z -242.561,A -90.000,B 90.000,C 0.000} C_DIS
LIN {X -144.015,Y -96.438,Z -242.561,A -90.000,B 90.000,C 0.000} C_DIS
LIN {X -144.015,Y -83.938,Z -242.561,A -90.000,B 90.000,C 0.000} C_DIS
LIN {X -144.015,Y -71.438,Z -242.561,A -90.000,B 90.000,C 0.000} C_DIS
LIN {X 144.015,Y -71.438,Z -242.561,A -90.000,B 90.000,C 0.000} C_DIS
LIN {X 144.015,Y -71.438,Z -235.012,A -90.000,B 90.000,C 0.000} C_DIS
LIN {X -144.015,Y -71.438,Z -235.012,A -90.000,B 90.000,C 0.000} C_DIS
LIN {X -144.015,Y -71.438,Z -227.464,A -90.000,B 90.000,C 0.000} C_DIS
LIN {X 144.015,Y -71.438,Z -227.464,A -90.000,B 90.000,C 0.000} C_DIS
LIN {X 144.015,Y -71.438,Z -219.915,A -90.000,B 90.000,C 0.000} C_DIS
LIN {X -144.015,Y -71.438,Z -219.915,A -90.000,B 90.000,C 0.000} C_DIS
LIN {X -144.015,Y -71.438,Z -212.366,A -90.000,B 90.000,C 0.000} C_DIS
LIN {X 144.015,Y -71.438,Z -212.366,A -90.000,B 90.000,C 0.000} C_DIS
LIN {X 144.015,Y -71.438,Z -204.817,A -90.000,B 90.000,C 0.000} C_DIS
LIN {X -144.015,Y -71.438,Z -204.817,A -90.000,B 90.000,C 0.000} C_DIS
LIN {X -144.015,Y -71.438,Z -197.269,A -90.000,B 90.000,C 0.000} C_DIS
LIN {X 144.015,Y -71.438,Z -197.269,A -90.000,B 90.000,C 0.000} C_DIS
LIN {X 144.015,Y -71.438,Z -189.720,A -90.000,B 90.000,C 0.000} C_DIS
LIN {X -144.015,Y -71.438,Z -189.720,A -90.000,B 90.000,C 0.000} C_DIS
LIN {X -144.015,Y -71.438,Z -182.171,A -90.000,B 90.000,C 0.000} C_DIS
LIN {X 144.015,Y -71.438,Z -182.171,A -90.000,B 90.000,C 0.000} C_DIS
LIN {X 144.015,Y -71.438,Z -174.622,A -90.000,B 90.000,C 0.000} C_DIS
LIN {X -144.015,Y -71.438,Z -174.622,A -90.000,B 90.000,C 0.000} C_DIS
LIN {X -144.015,Y -71.438,Z -167.073,A -90.000,B 90.000,C 0.000} C_DIS
LIN {X 144.015,Y -71.438,Z -167.073,A -90.000,B 90.000,C 0.000} C_DIS
LIN {X 144.015,Y -71.438,Z -159.525,A -90.000,B 90.000,C 0.000} C_DIS
LIN {X -144.015,Y -71.438,Z -159.525,A -90.000,B 90.000,C 0.000} C_DIS
LIN {X -144.015,Y -71.438,Z -151.976,A -90.000,B 90.000,C 0.000} C_DIS
LIN {X 144.015,Y -71.438,Z -151.976,A -90.000,B 90.000,C 0.000} C_DIS
LIN {X 144.015,Y -71.438,Z -144.427,A -90.000,B 90.000,C 0.000} C_DIS
LIN {X -144.015,Y -71.438,Z -144.427,A -90.000,B 90.000,C 0.000} C_DIS
LIN {X -144.015,Y -71.438,Z -136.878,A -90.000,B 90.000,C 0.000} C_DIS
LIN {X 144.015,Y -71.438,Z -136.878,A -90.000,B 90.000,C 0.000} C_DIS
LIN {X 144.015,Y -71.438,Z -129.329,A -90.000,B 90.000,C 0.000} C_DIS
LIN {X -144.015,Y -71.438,Z -129.329,A -90.000,B 90.000,C 0.000} C_DIS
LIN {X -144.015,Y -71.438,Z -121.781,A -90.000,B 90.000,C 0.000} C_DIS
LIN {X 144.015,Y -71.438,Z -121.781,A -90.000,B 90.000,C 0.000} C_DIS
LIN {X 144.015,Y -71.438,Z -114.232,A -90.000,B 90.000,C 0.000} C_DIS
LIN {X -144.015,Y -71.438,Z -114.232,A -90.000,B 90.000,C 0.000} C_DIS
LIN {X -144.015,Y -71.438,Z -106.683,A -90.000,B 90.000,C 0.000} C_DIS
LIN {X 144.015,Y -71.438,Z -106.683,A -90.000,B 90.000,C 0.000} C_DIS
LIN {X 144.015,Y -71.438,Z -99.134,A -90.000,B 90.000,C 0.000} C_DIS
LIN {X -144.015,Y -71.438,Z -99.134,A -90.000,B 90.000,C 0.000} C_DIS
LIN {X -144.015,Y -71.438,Z -91.586,A -90.000,B 90.000,C 0.000} C_DIS
LIN {X 144.015,Y -71.438,Z -91.586,A -90.000,B 90.000,C 0.000} C_DIS
LIN {X 144.015,Y -71.438,Z -84.037,A -90.000,B 90.000,C 0.000} C_DIS
LIN {X -144.015,Y -71.438,Z -84.037,A -90.000,B 90.000,C 0.000} C_DIS
LIN {X -144.015,Y -71.438,Z -76.488,A -90.000,B 90.000,C 0.000} C_DIS
LIN {X 144.015,Y -71.438,Z -76.488,A -90.000,B 90.000,C 0.000} C_DIS
LIN {X 144.015,Y -71.438,Z -68.939,A -90.000,B 90.000,C 0.000} C_DIS
LIN {X -144.015,Y -71.438,Z -68.939,A -90.000,B 90.000,C 0.000} C_DIS
LIN {X -144.015,Y -71.438,Z -61.390,A -90.000,B 90.000,C 0.000} C_DIS
LIN {X 144.015,Y -71.438,Z -61.390,A -90.000,B 90.000,C 0.000} C_DIS
LIN {X 144.015,Y -71.438,Z -53.842,A -90.000,B 90.000,C 0.000} C_DIS
LIN {X -144.015,Y -71.438,Z -53.842,A -90.000,B 90.000,C 0.000} C_DIS
LIN {X -144.015,Y -71.438,Z -46.293,A -90.000,B 90.000,C 0.000} C_DIS
LIN {X 144.015,Y -71.438,Z -46.293,A -90.000,B 90.000,C 0.000} C_DIS
LIN {X 144.015,Y -71.438,Z -38.744,A -90.000,B 90.000,C 0.000} C_DIS
LIN {X -144.015,Y -71.438,Z -38.744,A -90.000,B 90.000,C 0.000} C_DIS
LIN {X -144.015,Y -71.438,Z -31.195,A -90.000,B 90.000,C 0.000} C_DIS
LIN {X 144.015,Y -71.438,Z -31.195,A -90.000,B 90.000,C 0.000} C_DIS
LIN {X 144.015,Y -71.438,Z -23.646,A -90.000,B 90.000,C 0.000} C_DIS
LIN {X -144.015,Y -71.438,Z -23.646,A -90.000,B 90.000,C 0.000} C_DIS
LIN {X -144.015,Y -71.438,Z -16.098,A -90.000,B 90.000,C 0.000} C_DIS
LIN {X 144.015,Y -71.438,Z -16.098,A -90.000,B 90.000,C 0.000} C_DIS
LIN {X 144.015,Y -71.438,Z -8.549,A -90.000,B 90.000,C 0.000} C_DIS
LIN {X -144.015,Y -71.438,Z -8.549,A -90.000,B 90.000,C 0.000} C_DIS
LIN {X -144.015,Y -71.438,Z -1.000,A -90.000,B 90.000,C 0.000} C_DIS
LIN {X 144.015,Y -71.438,Z -1.000,A -90.000,B 90.000,C 0.000} C_DIS
LIN {X 145.015,Y -71.438,Z 0.000,A -90.000,B 90.000,C 0.000} C_DIS
LIN {X -145.015,Y -71.438,Z 0.000,A -90.000,B 90.000,C 0.000} C_DIS
LIN {X -145.015,Y -71.438,Z -243.561,A -90.000,B 90.000,C 0.000} C_DIS
LIN {X 145.015,Y -71.438,Z -243.561,A -90.000,B 90.000,C 0.000} C_DIS
LIN {X 145.015,Y -71.438,Z 0.000,A -90.000,B 90.000,C 0.000} C_DIS
LIN {X 145.015,Y -83.938,Z 0.000,A -90.000,B 90.000,C 0.000} C_DIS
LIN {X 145.015,Y -96.438,Z 0.000,A -90.000,B 90.000,C 0.000} C_DIS
LIN {X -144.015,Y -96.438,Z -242.561,A -90.000,B 90.000,C 0.000} C_DIS
LIN {X -144.015,Y -89.294,Z -242.561,A -90.000,B 90.000,C 0.000} C_DIS
LIN {X -144.015,Y -76.794,Z -242.561,A -90.000,B 90.000,C 0.000} C_DIS
LIN {X -144.015,Y -64.294,Z -242.561,A -90.000,B 90.000,C 0.000} C_DIS
LIN {X 144.015,Y -64.294,Z -242.561,A -90.000,B 90.000,C 0.000} C_DIS
LIN {X 144.015,Y -64.294,Z -235.012,A -90.000,B 90.000,C 0.000} C_DIS
LIN {X -144.015,Y -64.294,Z -235.012,A -90.000,B 90.000,C 0.000} C_DIS
LIN {X -144.015,Y -64.294,Z -227.464,A -90.000,B 90.000,C 0.000} C_DIS
LIN {X 144.015,Y -64.294,Z -227.464,A -90.000,B 90.000,C 0.000} C_DIS
LIN {X 144.015,Y -64.294,Z -219.915,A -90.000,B 90.000,C 0.000} C_DIS
LIN {X -144.015,Y -64.294,Z -219.915,A -90.000,B 90.000,C 0.000} C_DIS
LIN {X -144.015,Y -64.294,Z -212.366,A -90.000,B 90.000,C 0.000} C_DIS
LIN {X 144.015,Y -64.294,Z -212.366,A -90.000,B 90.000,C 0.000} C_DIS
LIN {X 144.015,Y -64.294,Z -204.817,A -90.000,B 90.000,C 0.000} C_DIS
LIN {X -144.015,Y -64.294,Z -204.817,A -90.000,B 90.000,C 0.000} C_DIS
LIN {X -144.015,Y -64.294,Z -197.269,A -90.000,B 90.000,C 0.000} C_DIS
LIN {X 144.015,Y -64.294,Z -197.269,A -90.000,B 90.000,C 0.000} C_DIS
LIN {X 144.015,Y -64.294,Z -189.720,A -90.000,B 90.000,C 0.000} C_DIS
LIN {X -144.015,Y -64.294,Z -189.720,A -90.000,B 90.000,C 0.000} C_DIS
LIN {X -144.015,Y -64.294,Z -182.171,A -90.000,B 90.000,C 0.000} C_DIS
LIN {X 144.015,Y -64.294,Z -182.171,A -90.000,B 90.000,C 0.000} C_DIS
LIN {X 144.015,Y -64.294,Z -174.622,A -90.000,B 90.000,C 0.000} C_DIS
LIN {X -144.015,Y -64.294,Z -174.622,A -90.000,B 90.000,C 0.000} C_DIS
LIN {X -144.015,Y -64.294,Z -167.073,A -90.000,B 90.000,C 0.000} C_DIS
LIN {X 144.015,Y -64.294,Z -167.073,A -90.000,B 90.000,C 0.000} C_DIS
LIN {X 144.015,Y -64.294,Z -159.525,A -90.000,B 90.000,C 0.000} C_DIS
LIN {X -144.015,Y -64.294,Z -159.525,A -90.000,B 90.000,C 0.000} C_DIS
LIN {X -144.015,Y -64.294,Z -151.976,A -90.000,B 90.000,C 0.000} C_DIS
LIN {X 144.015,Y -64.294,Z -151.976,A -90.000,B 90.000,C 0.000} C_DIS
LIN {X 144.015,Y -64.294,Z -144.427,A -90.000,B 90.000,C 0.000} C_DIS
LIN {X -144.015,Y -64.294,Z -144.427,A -90.000,B 90.000,C 0.000} C_DIS
LIN {X -144.015,Y -64.294,Z -136.878,A -90.000,B 90.000,C 0.000} C_DIS
LIN {X 144.015,Y -64.294,Z -136.878,A -90.000,B 90.000,C 0.000} C_DIS
LIN {X 144.015,Y -64.294,Z -129.329,A -90.000,B 90.000,C 0.000} C_DIS
LIN {X -144.015,Y -64.294,Z -129.329,A -90.000,B 90.000,C 0.000} C_DIS
LIN {X -144.015,Y -64.294,Z -121.781,A -90.000,B 90.000,C 0.000} C_DIS
LIN {X 144.015,Y -64.294,Z -121.781,A -90.000,B 90.000,C 0.000} C_DIS
LIN {X 144.015,Y -64.294,Z -114.232,A -90.000,B 90.000,C 0.000} C_DIS
LIN {X -144.015,Y -64.294,Z -114.232,A -90.000,B 90.000,C 0.000} C_DIS
LIN {X -144.015,Y -64.294,Z -106.683,A -90.000,B 90.000,C 0.000} C_DIS
LIN {X 144.015,Y -64.294,Z -106.683,A -90.000,B 90.000,C 0.000} C_DIS
LIN {X 144.015,Y -64.294,Z -99.134,A -90.000,B 90.000,C 0.000} C_DIS
LIN {X -144.015,Y -64.294,Z -99.134,A -90.000,B 90.000,C 0.000} C_DIS
LIN {X -144.015,Y -64.294,Z -91.586,A -90.000,B 90.000,C 0.000} C_DIS
LIN {X 144.015,Y -64.294,Z -91.586,A -90.000,B 90.000,C 0.000} C_DIS
LIN {X 144.015,Y -64.294,Z -84.037,A -90.000,B 90.000,C 0.000} C_DIS
LIN {X -144.015,Y -64.294,Z -84.037,A -90.000,B 90.000,C 0.000} C_DIS
LIN {X -144.015,Y -64.294,Z -76.488,A -90.000,B 90.000,C 0.000} C_DIS
LIN {X 144.015,Y -64.294,Z -76.488,A -90.000,B 90.000,C 0.000} C_DIS
LIN {X 144.015,Y -64.294,Z -68.939,A -90.000,B 90.000,C 0.000} C_DIS
LIN {X -144.015,Y -64.294,Z -68.939,A -90.000,B 90.000,C 0.000} C_DIS
LIN {X -144.015,Y -64.294,Z -61.390,A -90.000,B 90.000,C 0.000} C_DIS
LIN {X 144.015,Y -64.294,Z -61.390,A -90.000,B 90.000,C 0.000} C_DIS
LIN {X 144.015,Y -64.294,Z -53.842,A -90.000,B 90.000,C 0.000} C_DIS
LIN {X -144.015,Y -64.294,Z -53.842,A -90.000,B 90.000,C 0.000} C_DIS
LIN {X -144.015,Y -64.294,Z -46.293,A -90.000,B 90.000,C 0.000} C_DIS
LIN {X 144.015,Y -64.294,Z -46.293,A -90.000,B 90.000,C 0.000} C_DIS
LIN {X 144.015,Y -64.294,Z -38.744,A -90.000,B 90.000,C 0.000} C_DIS
LIN {X -144.015,Y -64.294,Z -38.744,A -90.000,B 90.000,C 0.000} C_DIS
LIN {X -144.015,Y -64.294,Z -31.195,A -90.000,B 90.000,C 0.000} C_DIS
LIN {X 144.015,Y -64.294,Z -31.195,A -90.000,B 90.000,C 0.000} C_DIS
LIN {X 144.015,Y -64.294,Z -23.646,A -90.000,B 90.000,C 0.000} C_DIS
LIN {X -144.015,Y -64.294,Z -23.646,A -90.000,B 90.000,C 0.000} C_DIS
LIN {X -144.015,Y -64.294,Z -16.098,A -90.000,B 90.000,C 0.000} C_DIS
LIN {X 144.015,Y -64.294,Z -16.098,A -90.000,B 90.000,C 0.000} C_DIS
LIN {X 144.015,Y -64.294,Z -8.549,A -90.000,B 90.000,C 0.000} C_DIS
LIN {X -144.015,Y -64.294,Z -8.549,A -90.000,B 90.000,C 0.000} C_DIS
LIN {X -144.015,Y -64.294,Z -1.000,A -90.000,B 90.000,C 0.000} C_DIS
LIN {X 144.015,Y -64.294,Z -1.000,A -90.000,B 90.000,C 0.000} C_DIS
LIN {X 145.015,Y -64.294,Z 0.000,A -90.000,B 90.000,C 0.000} C_DIS
LIN {X -145.015,Y -64.294,Z 0.000,A -90.000,B 90.000,C 0.000} C_DIS
LIN {X -145.015,Y -64.294,Z -243.561,A -90.000,B 90.000,C 0.000} C_DIS
LIN {X 145.015,Y -64.294,Z -243.561,A -90.000,B 90.000,C 0.000} C_DIS
LIN {X 145.015,Y -64.294,Z 0.000,A -90.000,B 90.000,C 0.000} C_DIS
LIN {X 145.015,Y -76.794,Z 0.000,A -90.000,B 90.000,C 0.000} C_DIS
LIN {X 145.015,Y -89.294,Z 0.000,A -90.000,B 90.000,C 0.000} C_DIS
LIN {X -144.015,Y -89.294,Z -242.561,A -90.000,B 90.000,C 0.000} C_DIS
LIN {X -144.015,Y -82.150,Z -242.561,A -90.000,B 90.000,C 0.000} C_DIS
LIN {X -144.015,Y -69.650,Z -242.561,A -90.000,B 90.000,C 0.000} C_DIS
LIN {X -144.015,Y -57.150,Z -242.561,A -90.000,B 90.000,C 0.000} C_DIS
LIN {X 144.015,Y -57.150,Z -242.561,A -90.000,B 90.000,C 0.000} C_DIS
LIN {X 144.015,Y -57.150,Z -235.012,A -90.000,B 90.000,C 0.000} C_DIS
LIN {X -144.015,Y -57.150,Z -235.012,A -90.000,B 90.000,C 0.000} C_DIS
LIN {X -144.015,Y -57.150,Z -227.464,A -90.000,B 90.000,C 0.000} C_DIS
LIN {X 144.015,Y -57.150,Z -227.464,A -90.000,B 90.000,C 0.000} C_DIS
LIN {X 144.015,Y -57.150,Z -219.915,A -90.000,B 90.000,C 0.000} C_DIS
LIN {X -144.015,Y -57.150,Z -219.915,A -90.000,B 90.000,C 0.000} C_DIS
LIN {X -144.015,Y -57.150,Z -212.366,A -90.000,B 90.000,C 0.000} C_DIS
LIN {X 144.015,Y -57.150,Z -212.366,A -90.000,B 90.000,C 0.000} C_DIS
LIN {X 144.015,Y -57.150,Z -204.817,A -90.000,B 90.000,C 0.000} C_DIS
LIN {X -144.015,Y -57.150,Z -204.817,A -90.000,B 90.000,C 0.000} C_DIS
LIN {X -144.015,Y -57.150,Z -197.269,A -90.000,B 90.000,C 0.000} C_DIS
LIN {X 144.015,Y -57.150,Z -197.269,A -90.000,B 90.000,C 0.000} C_DIS
LIN {X 144.015,Y -57.150,Z -189.720,A -90.000,B 90.000,C 0.000} C_DIS
LIN {X -144.015,Y -57.150,Z -189.720,A -90.000,B 90.000,C 0.000} C_DIS
LIN {X -144.015,Y -57.150,Z -182.171,A -90.000,B 90.000,C 0.000} C_DIS
LIN {X 144.015,Y -57.150,Z -182.171,A -90.000,B 90.000,C 0.000} C_DIS
LIN {X 144.015,Y -57.150,Z -174.622,A -90.000,B 90.000,C 0.000} C_DIS
LIN {X -144.015,Y -57.150,Z -174.622,A -90.000,B 90.000,C 0.000} C_DIS
LIN {X -144.015,Y -57.150,Z -167.073,A -90.000,B 90.000,C 0.000} C_DIS
LIN {X 144.015,Y -57.150,Z -167.073,A -90.000,B 90.000,C 0.000} C_DIS
LIN {X 144.015,Y -57.150,Z -159.525,A -90.000,B 90.000,C 0.000} C_DIS
LIN {X -144.015,Y -57.150,Z -159.525,A -90.000,B 90.000,C 0.000} C_DIS
LIN {X -144.015,Y -57.150,Z -151.976,A -90.000,B 90.000,C 0.000} C_DIS
LIN {X 144.015,Y -57.150,Z -151.976,A -90.000,B 90.000,C 0.000} C_DIS
LIN {X 144.015,Y -57.150,Z -144.427,A -90.000,B 90.000,C 0.000} C_DIS
LIN {X -144.015,Y -57.150,Z -144.427,A -90.000,B 90.000,C 0.000} C_DIS
LIN {X -144.015,Y -57.150,Z -136.878,A -90.000,B 90.000,C 0.000} C_DIS
LIN {X 144.015,Y -57.150,Z -136.878,A -90.000,B 90.000,C 0.000} C_DIS
LIN {X 144.015,Y -57.150,Z -129.329,A -90.000,B 90.000,C 0.000} C_DIS
LIN {X -144.015,Y -57.150,Z -129.329,A -90.000,B 90.000,C 0.000} C_DIS
LIN {X -144.015,Y -57.150,Z -121.781,A -90.000,B 90.000,C 0.000} C_DIS
LIN {X 144.015,Y -57.150,Z -121.781,A -90.000,B 90.000,C 0.000} C_DIS
LIN {X 144.015,Y -57.150,Z -114.232,A -90.000,B 90.000,C 0.000} C_DIS
LIN {X -144.015,Y -57.150,Z -114.232,A -90.000,B 90.000,C 0.000} C_DIS
LIN {X -144.015,Y -57.150,Z -106.683,A -90.000,B 90.000,C 0.000} C_DIS
LIN {X 144.015,Y -57.150,Z -106.683,A -90.000,B 90.000,C 0.000} C_DIS
LIN {X 144.015,Y -57.150,Z -99.134,A -90.000,B 90.000,C 0.000} C_DIS
LIN {X -144.015,Y -57.150,Z -99.134,A -90.000,B 90.000,C 0.000} C_DIS
LIN {X -144.015,Y -57.150,Z -91.586,A -90.000,B 90.000,C 0.000} C_DIS
LIN {X 144.015,Y -57.150,Z -91.586,A -90.000,B 90.000,C 0.000} C_DIS
LIN {X 144.015,Y -57.150,Z -84.037,A -90.000,B 90.000,C 0.000} C_DIS
LIN {X -144.015,Y -57.150,Z -84.037,A -90.000,B 90.000,C 0.000} C_DIS
LIN {X -144.015,Y -57.150,Z -76.488,A -90.000,B 90.000,C 0.000} C_DIS
LIN {X 144.015,Y -57.150,Z -76.488,A -90.000,B 90.000,C 0.000} C_DIS
LIN {X 144.015,Y -57.150,Z -68.939,A -90.000,B 90.000,C 0.000} C_DIS
LIN {X -144.015,Y -57.150,Z -68.939,A -90.000,B 90.000,C 0.000} C_DIS
LIN {X -144.015,Y -57.150,Z -61.390,A -90.000,B 90.000,C 0.000} C_DIS
LIN {X 144.015,Y -57.150,Z -61.390,A -90.000,B 90.000,C 0.000} C_DIS
LIN {X 144.015,Y -57.150,Z -53.842,A -90.000,B 90.000,C 0.000} C_DIS
LIN {X -144.015,Y -57.150,Z -53.842,A -90.000,B 90.000,C 0.000} C_DIS
LIN {X -144.015,Y -57.150,Z -46.293,A -90.000,B 90.000,C 0.000} C_DIS
LIN {X 144.015,Y -57.150,Z -46.293,A -90.000,B 90.000,C 0.000} C_DIS
LIN {X 144.015,Y -57.150,Z -38.744,A -90.000,B 90.000,C 0.000} C_DIS
LIN {X -144.015,Y -57.150,Z -38.744,A -90.000,B 90.000,C 0.000} C_DIS
LIN {X -144.015,Y -57.150,Z -31.195,A -90.000,B 90.000,C 0.000} C_DIS
LIN {X 144.015,Y -57.150,Z -31.195,A -90.000,B 90.000,C 0.000} C_DIS
LIN {X 144.015,Y -57.150,Z -23.646,A -90.000,B 90.000,C 0.000} C_DIS
LIN {X -144.015,Y -57.150,Z -23.646,A -90.000,B 90.000,C 0.000} C_DIS
LIN {X -144.015,Y -57.150,Z -16.098,A -90.000,B 90.000,C 0.000} C_DIS
LIN {X 144.015,Y -57.150,Z -16.098,A -90.000,B 90.000,C 0.000} C_DIS
LIN {X 144.015,Y -57.150,Z -8.549,A -90.000,B 90.000,C 0.000} C_DIS
LIN {X -144.015,Y -57.150,Z -8.549,A -90.000,B 90.000,C 0.000} C_DIS
LIN {X -144.015,Y -57.150,Z -1.000,A -90.000,B 90.000,C 0.000} C_DIS
LIN {X 144.015,Y -57.150,Z -1.000,A -90.000,B 90.000,C 0.000} C_DIS
LIN {X 145.015,Y -57.150,Z 0.000,A -90.000,B 90.000,C 0.000} C_DIS
LIN {X -145.015,Y -57.150,Z 0.000,A -90.000,B 90.000,C 0.000} C_DIS
LIN {X -145.015,Y -57.150,Z -243.561,A -90.000,B 90.000,C 0.000} C_DIS
LIN {X 145.015,Y -57.150,Z -243.561,A -90.000,B 90.000,C 0.000} C_DIS
LIN {X 145.015,Y -57.150,Z 0.000,A -90.000,B 90.000,C 0.000} C_DIS
LIN {X 145.015,Y -69.650,Z 0.000,A -90.000,B 90.000,C 0.000} C_DIS
LIN {X 145.015,Y -82.150,Z 0.000,A -90.000,B 90.000,C 0.000} C_DIS
LIN {X -144.015,Y -82.150,Z -242.561,A -90.000,B 90.000,C 0.000} C_DIS
LIN {X -144.015,Y -75.006,Z -242.561,A -90.000,B 90.000,C 0.000} C_DIS
LIN {X -144.015,Y -62.506,Z -242.561,A -90.000,B 90.000,C 0.000} C_DIS
LIN {X -144.015,Y -50.006,Z -242.561,A -90.000,B 90.000,C 0.000} C_DIS
LIN {X -73.727,Y -50.006,Z -242.561,A -90.000,B 90.000,C 0.000} C_DIS
LIN {X -71.291,Y -50.006,Z -241.287,A -90.000,B 90.000,C 0.000} C_DIS
LIN {X -68.834,Y -50.006,Z -240.054,A -90.000,B 90.000,C 0.000} C_DIS
LIN {X -66.358,Y -50.006,Z -238.862,A -90.000,B 90.000,C 0.000} C_DIS
LIN {X -63.861,Y -50.006,Z -237.712,A -90.000,B 90.000,C 0.000} C_DIS
LIN {X -61.346,Y -50.006,Z -236.603,A -90.000,B 90.000,C 0.000} C_DIS
LIN {X -56.640,Y -50.006,Z -235.012,A -90.000,B 90.000,C 0.000} C_DIS
LIN {X -144.015,Y -50.006,Z -235.012,A -90.000,B 90.000,C 0.000} C_DIS
LIN {X -144.015,Y -50.006,Z -227.464,A -90.000,B 90.000,C 0.000} C_DIS
LIN {X 14.485,Y -50.006,Z -227.464,A -90.000,B 90.000,C 0.000} C_DIS
LIN {X 14.603,Y -50.006,Z -226.329,A -90.000,B 90.000,C 0.000} C_DIS
LIN {X 14.761,Y -50.006,Z -225.200,A -90.000,B 90.000,C 0.000} C_DIS
LIN {X 14.960,Y -50.006,Z -224.076,A -90.000,B 90.000,C 0.000} C_DIS
LIN {X 15.199,Y -50.006,Z -222.961,A -90.000,B 90.000,C 0.000} C_DIS
LIN {X 15.796,Y -50.006,Z -221.432,A -90.000,B 90.000,C 0.000} C_DIS
LIN {X 16.421,Y -50.006,Z -219.915,A -90.000,B 90.000,C 0.000} C_DIS
LIN {X -144.015,Y -50.006,Z -219.915,A -90.000,B 90.000,C 0.000} C_DIS
LIN {X -144.015,Y -50.006,Z -212.366,A -90.000,B 90.000,C 0.000} C_DIS
LIN {X 20.043,Y -50.006,Z -212.366,A -90.000,B 90.000,C 0.000} C_DIS
LIN {X 20.523,Y -50.006,Z -211.489,A -90.000,B 90.000,C 0.000} C_DIS
LIN {X 21.013,Y -50.006,Z -210.617,A -90.000,B 90.000,C 0.000} C_DIS
LIN {X 21.756,Y -50.006,Z -209.428,A -90.000,B 90.000,C 0.000} C_DIS
LIN {X 22.467,Y -50.006,Z -208.219,A -90.000,B 90.000,C 0.000} C_DIS
LIN {X 23.148,Y -50.006,Z -206.993,A -90.000,B 90.000,C 0.000} C_DIS
LIN {X 23.796,Y -50.006,Z -205.750,A -90.000,B 90.000,C 0.000} C_DIS
LIN {X 24.407,Y -50.006,Z -204.817,A -90.000,B 90.000,C 0.000} C_DIS
LIN {X -144.015,Y -50.006,Z -204.817,A -90.000,B 90.000,C 0.000} C_DIS
LIN {X -144.015,Y -50.006,Z -197.269,A -90.000,B 90.000,C 0.000} C_DIS
LIN {X 29.249,Y -50.006,Z -197.269,A -90.000,B 90.000,C 0.000} C_DIS
LIN {X 30.853,Y -50.006,Z -194.948,A -90.000,B 90.000,C 0.000} C_DIS
LIN {X 31.253,Y -50.006,Z -194.224,A -90.000,B 90.000,C 0.000} C_DIS
LIN {X 31.703,Y -50.006,Z -193.530,A -90.000,B 90.000,C 0.000} C_DIS
LIN {X 32.202,Y -50.006,Z -192.871,A -90.000,B 90.000,C 0.000} C_DIS
LIN {X 32.746,Y -50.006,Z -192.249,A -90.000,B 90.000,C 0.000} C_DIS
LIN {X 33.334,Y -50.006,Z -191.667,A -90.000,B 90.000,C 0.000} C_DIS
LIN {X 33.962,Y -50.006,Z -191.129,A -90.000,B 90.000,C 0.000} C_DIS
LIN {X 34.627,Y -50.006,Z -190.637,A -90.000,B 90.000,C 0.000} C_DIS
LIN {X 35.325,Y -50.006,Z -190.194,A -90.000,B 90.000,C 0.000} C_DIS
LIN {X 36.053,Y -50.006,Z -189.802,A -90.000,B 90.000,C 0.000} C_DIS
LIN {X 36.318,Y -50.006,Z -189.720,A -90.000,B 90.000,C 0.000} C_DIS
LIN {X -144.015,Y -50.006,Z -189.720,A -90.000,B 90.000,C 0.000} C_DIS
LIN {X -144.015,Y -50.006,Z -182.171,A -90.000,B 90.000,C 0.000} C_DIS
LIN {X 144.015,Y -50.006,Z -182.171,A -90.000,B 90.000,C 0.000} C_DIS
LIN {X 144.015,Y -50.006,Z -174.622,A -90.000,B 90.000,C 0.000} C_DIS
LIN {X -144.015,Y -50.006,Z -174.622,A -90.000,B 90.000,C 0.000} C_DIS
LIN {X -144.015,Y -50.006,Z -167.073,A -90.000,B 90.000,C 0.000} C_DIS
LIN {X 144.015,Y -50.006,Z -167.073,A -90.000,B 90.000,C 0.000} C_DIS
LIN {X 144.015,Y -50.006,Z -159.525,A -90.000,B 90.000,C 0.000} C_DIS
LIN {X -144.015,Y -50.006,Z -159.525,A -90.000,B 90.000,C 0.000} C_DIS
LIN {X -144.015,Y -50.006,Z -151.976,A -90.000,B 90.000,C 0.000} C_DIS
LIN {X 144.015,Y -50.006,Z -151.976,A -90.000,B 90.000,C 0.000} C_DIS
LIN {X 144.015,Y -50.006,Z -144.427,A -90.000,B 90.000,C 0.000} C_DIS
LIN {X 17.239,Y -50.006,Z -144.427,A -90.000,B 90.000,C 0.000} C_DIS
LIN {X 18.282,Y -50.006,Z -144.012,A -90.000,B 90.000,C 0.000} C_DIS
LIN {X 19.304,Y -50.006,Z -143.546,A -90.000,B 90.000,C 0.000} C_DIS
LIN {X 20.303,Y -50.006,Z -143.032,A -90.000,B 90.000,C 0.000} C_DIS
LIN {X 21.275,Y -50.006,Z -142.470,A -90.000,B 90.000,C 0.000} C_DIS
LIN {X 22.222,Y -50.006,Z -141.648,A -90.000,B 90.000,C 0.000} C_DIS
LIN {X 23.126,Y -50.006,Z -140.779,A -90.000,B 90.000,C 0.000} C_DIS
LIN {X 23.985,Y -50.006,Z -139.865,A -90.000,B 90.000,C 0.000} C_DIS
LIN {X 24.796,Y -50.006,Z -138.909,A -90.000,B 90.000,C 0.000} C_DIS
LIN {X 25.557,Y -50.006,Z -137.913,A -90.000,B 90.000,C 0.000} C_DIS
LIN {X 26.266,Y -50.006,Z -136.878,A -90.000,B 90.000,C 0.000} C_DIS
LIN {X 144.015,Y -50.006,Z -136.878,A -90.000,B 90.000,C 0.000} C_DIS
LIN {X 144.015,Y -50.006,Z -129.329,A -90.000,B 90.000,C 0.000} C_DIS
LIN {X 28.237,Y -50.006,Z -129.329,A -90.000,B 90.000,C 0.000} C_DIS
LIN {X 28.183,Y -50.006,Z -128.333,A -90.000,B 90.000,C 0.000} C_DIS
LIN {X 28.061,Y -50.006,Z -127.343,A -90.000,B 90.000,C 0.000} C_DIS
LIN {X 27.872,Y -50.006,Z -126.364,A -90.000,B 90.000,C 0.000} C_DIS
LIN {X 27.618,Y -50.006,Z -125.400,A -90.000,B 90.000,C 0.000} C_DIS
LIN {X 27.298,Y -50.006,Z -124.455,A -90.000,B 90.000,C 0.000} C_DIS
LIN {X 26.915,Y -50.006,Z -123.534,A -90.000,B 90.000,C 0.000} C_DIS
LIN {X 26.471,Y -50.006,Z -122.641,A -90.000,B 90.000,C 0.000} C_DIS
LIN {X 25.966,Y -50.006,Z -121.781,A -90.000,B 90.000,C 0.000} C_DIS
LIN {X 144.015,Y -50.006,Z -121.781,A -90.000,B 90.000,C 0.000} C_DIS
LIN {X 144.015,Y -50.006,Z -114.232,A -90.000,B 90.000,C 0.000} C_DIS
LIN {X -144.015,Y -50.006,Z -114.232,A -90.000,B 90.000,C 0.000} C_DIS
LIN {X -144.015,Y -50.006,Z -106.683,A -90.000,B 90.000,C 0.000} C_DIS
LIN {X 144.015,Y -50.006,Z -106.683,A -90.000,B 90.000,C 0.000} C_DIS
LIN {X 144.015,Y -50.006,Z -99.134,A -90.000,B 90.000,C 0.000} C_DIS
LIN {X -144.015,Y -50.006,Z -99.134,A -90.000,B 90.000,C 0.000} C_DIS
LIN {X -144.015,Y -50.006,Z -91.586,A -90.000,B 90.000,C 0.000} C_DIS
LIN {X 144.015,Y -50.006,Z -91.586,A -90.000,B 90.000,C 0.000} C_DIS
LIN {X 144.015,Y -50.006,Z -84.037,A -90.000,B 90.000,C 0.000} C_DIS
LIN {X -144.015,Y -50.006,Z -84.037,A -90.000,B 90.000,C 0.000} C_DIS
LIN {X -144.015,Y -50.006,Z -76.488,A -90.000,B 90.000,C 0.000} C_DIS
LIN {X 81.355,Y -50.006,Z -76.488,A -90.000,B 90.000,C 0.000} C_DIS
LIN {X 81.092,Y -50.006,Z -76.281,A -90.000,B 90.000,C 0.000} C_DIS
LIN {X 80.835,Y -50.006,Z -76.067,A -90.000,B 90.000,C 0.000} C_DIS
LIN {X 80.722,Y -50.006,Z -75.985,A -90.000,B 90.000,C 0.000} C_DIS
LIN {X 80.015,Y -50.006,Z -75.454,A -90.000,B 90.000,C 0.000} C_DIS
LIN {X 79.345,Y -50.006,Z -74.876,A -90.000,B 90.000,C 0.000} C_DIS
LIN {X 78.715,Y -50.006,Z -74.255,A -90.000,B 90.000,C 0.000} C_DIS
LIN {X 78.129,Y -50.006,Z -73.593,A -90.000,B 90.000,C 0.000} C_DIS
LIN {X 77.588,Y -50.006,Z -72.893,A -90.000,B 90.000,C 0.000} C_DIS
LIN {X 77.096,Y -50.006,Z -72.158,A -90.000,B 90.000,C 0.000} C_DIS
LIN {X 76.654,Y -50.006,Z -71.392,A -90.000,B 90.000,C 0.000} C_DIS
LIN {X 76.265,Y -50.006,Z -70.597,A -90.000,B 90.000,C 0.000} C_DIS
LIN {X 75.930,Y -50.006,Z -69.779,A -90.000,B 90.000,C 0.000} C_DIS
LIN {X 75.652,Y -50.006,Z -68.939,A -90.000,B 90.000,C 0.000} C_DIS
LIN {X -144.015,Y -50.006,Z -68.939,A -90.000,B 90.000,C 0.000} C_DIS
LIN {X -144.015,Y -50.006,Z -61.390,A -90.000,B 90.000,C 0.000} C_DIS
LIN {X 75.365,Y -50.006,Z -61.390,A -90.000,B 90.000,C 0.000} C_DIS
LIN {X 75.572,Y -50.006,Z -60.466,A -90.000,B 90.000,C 0.000} C_DIS
LIN {X 75.832,Y -50.006,Z -59.555,A -90.000,B 90.000,C 0.000} C_DIS
LIN {X 76.144,Y -50.006,Z -58.661,A -90.000,B 90.000,C 0.000} C_DIS
LIN {X 76.506,Y -50.006,Z -57.786,A -90.000,B 90.000,C 0.000} C_DIS
LIN {X 76.917,Y -50.006,Z -56.933,A -90.000,B 90.000,C 0.000} C_DIS
LIN {X 77.596,Y -50.006,Z -55.878,A -90.000,B 90.000,C 0.000} C_DIS
LIN {X 78.312,Y -50.006,Z -54.847,A -90.000,B 90.000,C 0.000} C_DIS
LIN {X 79.064,Y -50.006,Z -53.842,A -90.000,B 90.000,C 0.000} C_DIS
LIN {X -144.015,Y -50.006,Z -53.842,A -90.000,B 90.000,C 0.000} C_DIS
LIN {X -144.015,Y -50.006,Z -46.293,A -90.000,B 90.000,C 0.000} C_DIS
LIN {X 86.747,Y -50.006,Z -46.293,A -90.000,B 90.000,C 0.000} C_DIS
LIN {X 88.724,Y -50.006,Z -44.582,A -90.000,B 90.000,C 0.000} C_DIS
LIN {X 90.692,Y -50.006,Z -42.861,A -90.000,B 90.000,C 0.000} C_DIS
LIN {X 91.453,Y -50.006,Z -42.084,A -90.000,B 90.000,C 0.000} C_DIS
LIN {X 92.249,Y -50.006,Z -41.342,A -90.000,B 90.000,C 0.000} C_DIS
LIN {X 93.076,Y -50.006,Z -40.635,A -90.000,B 90.000,C 0.000} C_DIS
LIN {X 93.933,Y -50.006,Z -39.966,A -90.000,B 90.000,C 0.000} C_DIS
LIN {X 94.820,Y -50.006,Z -39.335,A -90.000,B 90.000,C 0.000} C_DIS
LIN {X 95.733,Y -50.006,Z -38.744,A -90.000,B 90.000,C 0.000} C_DIS
LIN {X -144.015,Y -50.006,Z -38.744,A -90.000,B 90.000,C 0.000} C_DIS
LIN {X -144.015,Y -50.006,Z -31.195,A -90.000,B 90.000,C 0.000} C_DIS
LIN {X 144.015,Y -50.006,Z -31.195,A -90.000,B 90.000,C 0.000} C_DIS
LIN {X 144.015,Y -50.006,Z -23.646,A -90.000,B 90.000,C 0.000} C_DIS
LIN {X -144.015,Y -50.006,Z -23.646,A -90.000,B 90.000,C 0.000} C_DIS
LIN {X -144.015,Y -50.006,Z -16.098,A -90.000,B 90.000,C 0.000} C_DIS
LIN {X 144.015,Y -50.006,Z -16.098,A -90.000,B 90.000,C 0.000} C_DIS
LIN {X 144.015,Y -50.006,Z -8.549,A -90.000,B 90.000,C 0.000} C_DIS
LIN {X -144.015,Y -50.006,Z -8.549,A -90.000,B 90.000,C 0.000} C_DIS
LIN {X -144.015,Y -50.006,Z -1.000,A -90.000,B 90.000,C 0.000} C_DIS
LIN {X 144.015,Y -50.006,Z -1.000,A -90.000,B 90.000,C 0.000} C_DIS
LIN {X 144.015,Y -50.006,Z -38.744,A -90.000,B 90.000,C 0.000} C_DIS
LIN {X 110.370,Y -50.006,Z -38.744,A -90.000,B 90.000,C 0.000} C_DIS
LIN {X 111.045,Y -50.006,Z -39.284,A -90.000,B 90.000,C 0.000} C_DIS
LIN {X 111.678,Y -50.006,Z -39.872,A -90.000,B 90.000,C 0.000} C_DIS
LIN {X 112.267,Y -50.006,Z -40.505,A -90.000,B 90.000,C 0.000} C_DIS
LIN {X 112.808,Y -50.006,Z -41.179,A -90.000,B 90.000,C 0.000} C_DIS
LIN {X 113.297,Y -50.006,Z -41.892,A -90.000,B 90.000,C 0.000} C_DIS
LIN {X 113.734,Y -50.006,Z -42.638,A -90.000,B 90.000,C 0.000} C_DIS
LIN {X 114.114,Y -50.006,Z -43.414,A -90.000,B 90.000,C 0.000} C_DIS
LIN {X 114.437,Y -50.006,Z -44.216,A -90.000,B 90.000,C 0.000} C_DIS
LIN {X 114.700,Y -50.006,Z -45.039,A -90.000,B 90.000,C 0.000} C_DIS
LIN {X 114.836,Y -50.006,Z -45.664,A -90.000,B 90.000,C 0.000} C_DIS
LIN {X 114.949,Y -50.006,Z -46.293,A -90.000,B 90.000,C 0.000} C_DIS
LIN {X 144.015,Y -50.006,Z -46.293,A -90.000,B 90.000,C 0.000} C_DIS
LIN {X 144.015,Y -50.006,Z -53.842,A -90.000,B 90.000,C 0.000} C_DIS
LIN {X 114.789,Y -50.006,Z -53.842,A -90.000,B 90.000,C 0.000} C_DIS
LIN {X 114.580,Y -50.006,Z -55.376,A -90.000,B 90.000,C 0.000} C_DIS
LIN {X 114.308,Y -50.006,Z -56.901,A -90.000,B 90.000,C 0.000} C_DIS
LIN {X 113.973,Y -50.006,Z -58.413,A -90.000,B 90.000,C 0.000} C_DIS
LIN {X 113.577,Y -50.006,Z -59.910,A -90.000,B 90.000,C 0.000} C_DIS
LIN {X 113.120,Y -50.006,Z -61.390,A -90.000,B 90.000,C 0.000} C_DIS
LIN {X 144.015,Y -50.006,Z -61.390,A -90.000,B 90.000,C 0.000} C_DIS
LIN {X 144.015,Y -50.006,Z -68.939,A -90.000,B 90.000,C 0.000} C_DIS
LIN {X 109.663,Y -50.006,Z -68.939,A -90.000,B 90.000,C 0.000} C_DIS
LIN {X 109.050,Y -50.006,Z -69.915,A -90.000,B 90.000,C 0.000} C_DIS
LIN {X 108.393,Y -50.006,Z -70.861,A -90.000,B 90.000,C 0.000} C_DIS
LIN {X 107.692,Y -50.006,Z -71.776,A -90.000,B 90.000,C 0.000} C_DIS
LIN {X 106.950,Y -50.006,Z -72.658,A -90.000,B 90.000,C 0.000} C_DIS
LIN {X 106.168,Y -50.006,Z -73.504,A -90.000,B 90.000,C 0.000} C_DIS
LIN {X 105.347,Y -50.006,Z -74.313,A -90.000,B 90.000,C 0.000} C_DIS
LIN {X 104.490,Y -50.006,Z -75.083,A -90.000,B 90.000,C 0.000} C_DIS
LIN {X 103.598,Y -50.006,Z -75.813,A -90.000,B 90.000,C 0.000} C_DIS
LIN {X 103.174,Y -50.006,Z -76.157,A -90.000,B 90.000,C 0.000} C_DIS
LIN {X 102.739,Y -50.006,Z -76.488,A -90.000,B 90.000,C 0.000} C_DIS
LIN {X 144.015,Y -50.006,Z -76.488,A -90.000,B 90.000,C 0.000} C_DIS
LIN {X 144.015,Y -50.006,Z -189.720,A -90.000,B 90.000,C 0.000} C_DIS
LIN {X 51.708,Y -50.006,Z -189.720,A -90.000,B 90.000,C 0.000} C_DIS
LIN {X 52.332,Y -50.006,Z -190.295,A -90.000,B 90.000,C 0.000} C_DIS
LIN {X 52.907,Y -50.006,Z -190.919,A -90.000,B 90.000,C 0.000} C_DIS
LIN {X 53.430,Y -50.006,Z -191.586,A -90.000,B 90.000,C 0.000} C_DIS
LIN {X 53.898,Y -50.006,Z -192.294,A -90.000,B 90.000,C 0.000} C_DIS
LIN {X 54.307,Y -50.006,Z -193.037,A -90.000,B 90.000,C 0.000} C_DIS
LIN {X 54.655,Y -50.006,Z -193.811,A -90.000,B 90.000,C 0.000} C_DIS
LIN {X 54.940,Y -50.006,Z -194.610,A -90.000,B 90.000,C 0.000} C_DIS
LIN {X 55.159,Y -50.006,Z -195.429,A -90.000,B 90.000,C 0.000} C_DIS
LIN {X 55.312,Y -50.006,Z -196.264,A -90.000,B 90.000,C 0.000} C_DIS
LIN {X 55.370,Y -50.006,Z -197.269,A -90.000,B 90.000,C 0.000} C_DIS
LIN {X 144.015,Y -50.006,Z -197.269,A -90.000,B 90.000,C 0.000} C_DIS
LIN {X 144.015,Y -50.006,Z -204.817,A -90.000,B 90.000,C 0.000} C_DIS
LIN {X 55.846,Y -50.006,Z -204.817,A -90.000,B 90.000,C 0.000} C_DIS
LIN {X 55.648,Y -50.006,Z -206.262,A -90.000,B 90.000,C 0.000} C_DIS
LIN {X 55.391,Y -50.006,Z -207.697,A -90.000,B 90.000,C 0.000} C_DIS
LIN {X 55.074,Y -50.006,Z -209.120,A -90.000,B 90.000,C 0.000} C_DIS
LIN {X 54.699,Y -50.006,Z -210.530,A -90.000,B 90.000,C 0.000} C_DIS
LIN {X 54.266,Y -50.006,Z -211.922,A -90.000,B 90.000,C 0.000} C_DIS
LIN {X 54.170,Y -50.006,Z -212.366,A -90.000,B 90.000,C 0.000} C_DIS
LIN {X 144.015,Y -50.006,Z -212.366,A -90.000,B 90.000,C 0.000} C_DIS
LIN {X 144.015,Y -50.006,Z -219.915,A -90.000,B 90.000,C 0.000} C_DIS
LIN {X 52.176,Y -50.006,Z -219.915,A -90.000,B 90.000,C 0.000} C_DIS
LIN {X 51.675,Y -50.006,Z -221.484,A -90.000,B 90.000,C 0.000} C_DIS
LIN {X 51.147,Y -50.006,Z -223.043,A -90.000,B 90.000,C 0.000} C_DIS
LIN {X 50.591,Y -50.006,Z -224.593,A -90.000,B 90.000,C 0.000} C_DIS
LIN {X 49.943,Y -50.006,Z -226.038,A -90.000,B 90.000,C 0.000} C_DIS
LIN {X 49.255,Y -50.006,Z -227.464,A -90.000,B 90.000,C 0.000} C_DIS
LIN {X 144.015,Y -50.006,Z -227.464,A -90.000,B 90.000,C 0.000} C_DIS
LIN {X 144.015,Y -50.006,Z -235.012,A -90.000,B 90.000,C 0.000} C_DIS
LIN {X 44.277,Y -50.006,Z -235.012,A -90.000,B 90.000,C 0.000} C_DIS
LIN {X 43.106,Y -50.006,Z -236.219,A -90.000,B 90.000,C 0.000} C_DIS
LIN {X 41.905,Y -50.006,Z -237.395,A -90.000,B 90.000,C 0.000} C_DIS
LIN {X 40.674,Y -50.006,Z -238.539,A -90.000,B 90.000,C 0.000} C_DIS
LIN {X 39.414,Y -50.006,Z -239.652,A -90.000,B 90.000,C 0.000} C_DIS
LIN {X 38.246,Y -50.006,Z -240.362,A -90.000,B 90.000,C 0.000} C_DIS
LIN {X 37.058,Y -50.006,Z -241.037,A -90.000,B 90.000,C 0.000} C_DIS
LIN {X 35.850,Y -50.006,Z -241.676,A -90.000,B 90.000,C 0.000} C_DIS
LIN {X 34.624,Y -50.006,Z -242.279,A -90.000,B 90.000,C 0.000} C_DIS
LIN {X 34.351,Y -50.006,Z -242.424,A -90.000,B 90.000,C 0.000} C_DIS
LIN {X 34.073,Y -50.006,Z -242.561,A -90.000,B 90.000,C 0.000} C_DIS
LIN {X 144.015,Y -50.006,Z -242.561,A -90.000,B 90.000,C 0.000} C_DIS
LIN {X 0.925,Y -50.006,Z -144.427,A -90.000,B 90.000,C 0.000} C_DIS
LIN {X -144.015,Y -50.006,Z -144.427,A -90.000,B 90.000,C 0.000} C_DIS
LIN {X -144.015,Y -50.006,Z -136.878,A -90.000,B 90.000,C 0.000} C_DIS
LIN {X -5.888,Y -50.006,Z -136.878,A -90.000,B 90.000,C 0.000} C_DIS
LIN {X -6.190,Y -50.006,Z -136.005,A -90.000,B 90.000,C 0.000} C_DIS
LIN {X -6.447,Y -50.006,Z -135.117,A -90.000,B 90.000,C 0.000} C_DIS
LIN {X -6.661,Y -50.006,Z -134.218,A -90.000,B 90.000,C 0.000} C_DIS
LIN {X -6.830,Y -50.006,Z -133.310,A -90.000,B 90.000,C 0.000} C_DIS
LIN {X -6.951,Y -50.006,Z -132.518,A -90.000,B 90.000,C 0.000} C_DIS
LIN {X -7.012,Y -50.006,Z -131.720,A -90.000,B 90.000,C 0.000} C_DIS
LIN {X -7.012,Y -50.006,Z -130.919,A -90.000,B 90.000,C 0.000} C_DIS
LIN {X -6.952,Y -50.006,Z -130.121,A -90.000,B 90.000,C 0.000} C_DIS
LIN {X -6.830,Y -50.006,Z -129.329,A -90.000,B 90.000,C 0.000} C_DIS
LIN {X -144.015,Y -50.006,Z -129.329,A -90.000,B 90.000,C 0.000} C_DIS
LIN {X -144.015,Y -50.006,Z -121.781,A -90.000,B 90.000,C 0.000} C_DIS
LIN {X -2.598,Y -50.006,Z -121.781,A -90.000,B 90.000,C 0.000} C_DIS
LIN {X -2.955,Y -50.006,Z -122.223,A -90.000,B 90.000,C 0.000} C_DIS
LIN {X -3.290,Y -50.006,Z -122.682,A -90.000,B 90.000,C 0.000} C_DIS
LIN {X -3.602,Y -50.006,Z -123.156,A -90.000,B 90.000,C 0.000} C_DIS
LIN {X -4.225,Y -50.006,Z -123.925,A -90.000,B 90.000,C 0.000} C_DIS
LIN {X -4.801,Y -50.006,Z -124.730,A -90.000,B 90.000,C 0.000} C_DIS
LIN {X -5.329,Y -50.006,Z -125.567,A -90.000,B 90.000,C 0.000} C_DIS
LIN {X -5.807,Y -50.006,Z -126.433,A -90.000,B 90.000,C 0.000} C_DIS
LIN {X -6.233,Y -50.006,Z -127.326,A -90.000,B 90.000,C 0.000} C_DIS
LIN {X -6.496,Y -50.006,Z -128.041,A -90.000,B 90.000,C 0.000} C_DIS
LIN {X -6.707,Y -50.006,Z -128.774,A -90.000,B 90.000,C 0.000} C_DIS
LIN {X -6.865,Y -50.006,Z -129.519,A -90.000,B 90.000,C 0.000} C_DIS
LIN {X -6.968,Y -50.006,Z -130.274,A -90.000,B 90.000,C 0.000} C_DIS
LIN {X -7.016,Y -50.006,Z -131.035,A -90.000,B 90.000,C 0.000} C_DIS
LIN {X -7.009,Y -50.006,Z -131.797,A -90.000,B 90.000,C 0.000} C_DIS
LIN {X -6.947,Y -50.006,Z -132.557,A -90.000,B 90.000,C 0.000} C_DIS
LIN {X -6.830,Y -50.006,Z -133.310,A -90.000,B 90.000,C 0.000} C_DIS
LIN {X -6.676,Y -50.006,Z -134.145,A -90.000,B 90.000,C 0.000} C_DIS
LIN {X -6.485,Y -50.006,Z -134.972,A -90.000,B 90.000,C 0.000} C_DIS
LIN {X -6.256,Y -50.006,Z -135.790,A -90.000,B 90.000,C 0.000} C_DIS
LIN {X -5.991,Y -50.006,Z -136.596,A -90.000,B 90.000,C 0.000} C_DIS
LIN {X -28.529,Y -50.006,Z -235.012,A -90.000,B 90.000,C 0.000} C_DIS
LIN {X 15.405,Y -50.006,Z -235.012,A -90.000,B 90.000,C 0.000} C_DIS
LIN {X 15.516,Y -50.006,Z -235.556,A -90.000,B 90.000,C 0.000} C_DIS
LIN {X 15.815,Y -50.006,Z -236.328,A -90.000,B 90.000,C 0.000} C_DIS
LIN {X 16.174,Y -50.006,Z -237.073,A -90.000,B 90.000,C 0.000} C_DIS
LIN {X 16.590,Y -50.006,Z -237.789,A -90.000,B 90.000,C 0.000} C_DIS
LIN {X 17.061,Y -50.006,Z -238.469,A -90.000,B 90.000,C 0.000} C_DIS
LIN {X 17.584,Y -50.006,Z -239.110,A -90.000,B 90.000,C 0.000} C_DIS
LIN {X 18.156,Y -50.006,Z -239.708,A -90.000,B 90.000,C 0.000} C_DIS
LIN {X 18.774,Y -50.006,Z -240.259,A -90.000,B 90.000,C 0.000} C_DIS
LIN {X 19.432,Y -50.006,Z -240.761,A -90.000,B 90.000,C 0.000} C_DIS
LIN {X 20.128,Y -50.006,Z -241.208,A -90.000,B 90.000,C 0.000} C_DIS
LIN {X 20.857,Y -50.006,Z -241.600,A -90.000,B 90.000,C 0.000} C_DIS
LIN {X 21.614,Y -50.006,Z -241.933,A -90.000,B 90.000,C 0.000} C_DIS
LIN {X 22.396,Y -50.006,Z -242.206,A -90.000,B 90.000,C 0.000} C_DIS
LIN {X 23.196,Y -50.006,Z -242.417,A -90.000,B 90.000,C 0.000} C_DIS
LIN {X 23.942,Y -50.006,Z -242.561,A -90.000,B 90.000,C 0.000} C_DIS
LIN {X -21.138,Y -50.006,Z -242.561,A -90.000,B 90.000,C 0.000} C_DIS
LIN {X -21.687,Y -50.006,Z -243.561,A -90.000,B 90.000,C 0.000} C_DIS
LIN {X 145.015,Y -50.006,Z -243.561,A -90.000,B 90.000,C 0.000} C_DIS
LIN {X 145.015,Y -50.006,Z 0.000,A -90.000,B 90.000,C 0.000} C_DIS
LIN {X -145.015,Y -50.006,Z 0.000,A -90.000,B 90.000,C 0.000} C_DIS
LIN {X -145.015,Y -50.006,Z -243.561,A -90.000,B 90.000,C 0.000} C_DIS
LIN {X -73.477,Y -50.006,Z -243.561,A -90.000,B 90.000,C 0.000} C_DIS
LIN {X -71.020,Y -50.006,Z -242.272,A -90.000,B 90.000,C 0.000} C_DIS
LIN {X -68.543,Y -50.006,Z -241.025,A -90.000,B 90.000,C 0.000} C_DIS
LIN {X -66.044,Y -50.006,Z -239.820,A -90.000,B 90.000,C 0.000} C_DIS
LIN {X -63.525,Y -50.006,Z -238.657,A -90.000,B 90.000,C 0.000} C_DIS
LIN {X -60.987,Y -50.006,Z -237.538,A -90.000,B 90.000,C 0.000} C_DIS
LIN {X -50.864,Y -50.006,Z -234.116,A -90.000,B 90.000,C 0.000} C_DIS
LIN {X -49.212,Y -50.006,Z -233.768,A -90.000,B 90.000,C 0.000} C_DIS
LIN {X -47.553,Y -50.006,Z -233.461,A -90.000,B 90.000,C 0.000} C_DIS
LIN {X -45.886,Y -50.006,Z -233.193,A -90.000,B 90.000,C 0.000} C_DIS
LIN {X -44.214,Y -50.006,Z -232.966,A -90.000,B 90.000,C 0.000} C_DIS
LIN {X -42.536,Y -50.006,Z -232.780,A -90.000,B 90.000,C 0.000} C_DIS
LIN {X -41.081,Y -50.006,Z -232.779,A -90.000,B 90.000,C 0.000} C_DIS
LIN {X -39.627,Y -50.006,Z -232.831,A -90.000,B 90.000,C 0.000} C_DIS
LIN {X -38.176,Y -50.006,Z -232.937,A -90.000,B 90.000,C 0.000} C_DIS
LIN {X -36.730,Y -50.006,Z -233.095,A -90.000,B 90.000,C 0.000} C_DIS
LIN {X -35.290,Y -50.006,Z -233.306,A -90.000,B 90.000,C 0.000} C_DIS
LIN {X -34.070,Y -50.006,Z -233.672,A -90.000,B 90.000,C 0.000} C_DIS
LIN {X -32.867,Y -50.006,Z -234.094,A -90.000,B 90.000,C 0.000} C_DIS
LIN {X -31.685,Y -50.006,Z -234.569,A -90.000,B 90.000,C 0.000} C_DIS
LIN {X -30.526,Y -50.006,Z -235.098,A -90.000,B 90.000,C 0.000} C_DIS
LIN {X -29.392,Y -50.006,Z -235.679,A -90.000,B 90.000,C 0.000} C_DIS
LIN {X -28.285,Y -50.006,Z -236.311,A -90.000,B 90.000,C 0.000} C_DIS
LIN {X -27.322,Y -50.006,Z -237.080,A -90.000,B 90.000,C 0.000} C_DIS
LIN {X -26.395,Y -50.006,Z -237.891,A -90.000,B 90.000,C 0.000} C_DIS
LIN {X -25.506,Y -50.006,Z -238.744,A -90.000,B 90.000,C 0.000} C_DIS
LIN {X -24.656,Y -50.006,Z -239.636,A -90.000,B 90.000,C 0.000} C_DIS
LIN {X -23.848,Y -50.006,Z -240.566,A -90.000,B 90.000,C 0.000} C_DIS
LIN {X -23.083,Y -50.006,Z -241.531,A -90.000,B 90.000,C 0.000} C_DIS
LIN {X -22.362,Y -50.006,Z -242.530,A -90.000,B 90.000,C 0.000} C_DIS
LIN {X -21.687,Y -50.006,Z -243.561,A -90.000,B 90.000,C 0.000} C_DIS
LIN {X 16.482,Y -50.006,Z -235.289,A -90.000,B 90.000,C 0.000} C_DIS
LIN {X 16.155,Y -50.006,Z -233.612,A -90.000,B 90.000,C 0.000} C_DIS
LIN {X 15.868,Y -50.006,Z -231.928,A -90.000,B 90.000,C 0.000} C_DIS
LIN {X 15.621,Y -50.006,Z -230.238,A -90.000,B 90.000,C 0.000} C_DIS
LIN {X 15.413,Y -50.006,Z -228.542,A -90.000,B 90.000,C 0.000} C_DIS
LIN {X 15.513,Y -50.006,Z -227.209,A -90.000,B 90.000,C 0.000} C_DIS
LIN {X 15.671,Y -50.006,Z -225.881,A -90.000,B 90.000,C 0.000} C_DIS
LIN {X 15.886,Y -50.006,Z -224.562,A -90.000,B 90.000,C 0.000} C_DIS
LIN {X 16.158,Y -50.006,Z -223.253,A -90.000,B 90.000,C 0.000} C_DIS
LIN {X 16.980,Y -50.006,Z -221.174,A -90.000,B 90.000,C 0.000} C_DIS
LIN {X 17.854,Y -50.006,Z -219.118,A -90.000,B 90.000,C 0.000} C_DIS
LIN {X 18.781,Y -50.006,Z -217.084,A -90.000,B 90.000,C 0.000} C_DIS
LIN {X 19.759,Y -50.006,Z -215.074,A -90.000,B 90.000,C 0.000} C_DIS
LIN {X 20.789,Y -50.006,Z -213.091,A -90.000,B 90.000,C 0.000} C_DIS
LIN {X 21.869,Y -50.006,Z -211.134,A -90.000,B 90.000,C 0.000} C_DIS
LIN {X 22.614,Y -50.006,Z -209.940,A -90.000,B 90.000,C 0.000} C_DIS
LIN {X 23.328,Y -50.006,Z -208.728,A -90.000,B 90.000,C 0.000} C_DIS
LIN {X 24.011,Y -50.006,Z -207.499,A -90.000,B 90.000,C 0.000} C_DIS
LIN {X 24.663,Y -50.006,Z -206.252,A -90.000,B 90.000,C 0.000} C_DIS
LIN {X 28.609,Y -50.006,Z -200.232,A -90.000,B 90.000,C 0.000} C_DIS
LIN {X 29.124,Y -50.006,Z -199.206,A -90.000,B 90.000,C 0.000} C_DIS
LIN {X 31.716,Y -50.006,Z -195.459,A -90.000,B 90.000,C 0.000} C_DIS
LIN {X 32.124,Y -50.006,Z -194.716,A -90.000,B 90.000,C 0.000} C_DIS
LIN {X 32.591,Y -50.006,Z -194.007,A -90.000,B 90.000,C 0.000} C_DIS
LIN {X 33.114,Y -50.006,Z -193.339,A -90.000,B 90.000,C 0.000} C_DIS
LIN {X 33.688,Y -50.006,Z -192.715,A -90.000,B 90.000,C 0.000} C_DIS
LIN {X 34.310,Y -50.006,Z -192.138,A -90.000,B 90.000,C 0.000} C_DIS
LIN {X 34.977,Y -50.006,Z -191.614,A -90.000,B 90.000,C 0.000} C_DIS
LIN {X 35.684,Y -50.006,Z -191.145,A -90.000,B 90.000,C 0.000} C_DIS
LIN {X 36.426,Y -50.006,Z -190.734,A -90.000,B 90.000,C 0.000} C_DIS
LIN {X 37.829,Y -50.006,Z -190.277,A -90.000,B 90.000,C 0.000} C_DIS
LIN {X 39.219,Y -50.006,Z -189.782,A -90.000,B 90.000,C 0.000} C_DIS
LIN {X 40.595,Y -50.006,Z -189.249,A -90.000,B 90.000,C 0.000} C_DIS
LIN {X 41.955,Y -50.006,Z -188.678,A -90.000,B 90.000,C 0.000} C_DIS
LIN {X 42.753,Y -50.006,Z -188.457,A -90.000,B 90.000,C 0.000} C_DIS
LIN {X 43.567,Y -50.006,Z -188.307,A -90.000,B 90.000,C 0.000} C_DIS
LIN {X 44.391,Y -50.006,Z -188.227,A -90.000,B 90.000,C 0.000} C_DIS
LIN {X 45.219,Y -50.006,Z -188.220,A -90.000,B 90.000,C 0.000} C_DIS
LIN {X 46.045,Y -50.006,Z -188.284,A -90.000,B 90.000,C 0.000} C_DIS
LIN {X 46.862,Y -50.006,Z -188.420,A -90.000,B 90.000,C 0.000} C_DIS
LIN {X 47.664,Y -50.006,Z -188.627,A -90.000,B 90.000,C 0.000} C_DIS
LIN {X 48.444,Y -50.006,Z -188.902,A -90.000,B 90.000,C 0.000} C_DIS
LIN {X 49.199,Y -50.006,Z -189.244,A -90.000,B 90.000,C 0.000} C_DIS
LIN {X 49.920,Y -50.006,Z -189.650,A -90.000,B 90.000,C 0.000} C_DIS
LIN {X 50.604,Y -50.006,Z -190.117,A -90.000,B 90.000,C 0.000} C_DIS
LIN {X 51.244,Y -50.006,Z -190.642,A -90.000,B 90.000,C 0.000} C_DIS
LIN {X 51.836,Y -50.006,Z -191.221,A -90.000,B 90.000,C 0.000} C_DIS
LIN {X 52.376,Y -50.006,Z -191.849,A -90.000,B 90.000,C 0.000} C_DIS
LIN {X 52.859,Y -50.006,Z -192.521,A -90.000,B 90.000,C 0.000} C_DIS
LIN {X 53.282,Y -50.006,Z -193.233,A -90.000,B 90.000,C 0.000} C_DIS
LIN {X 53.642,Y -50.006,Z -193.979,A -90.000,B 90.000,C 0.000} C_DIS
LIN {X 53.936,Y -50.006,Z -194.753,A -90.000,B 90.000,C 0.000} C_DIS
LIN {X 54.161,Y -50.006,Z -195.550,A -90.000,B 90.000,C 0.000} C_DIS
LIN {X 54.316,Y -50.006,Z -196.363,A -90.000,B 90.000,C 0.000} C_DIS
LIN {X 54.568,Y -50.006,Z -200.514,A -90.000,B 90.000,C 0.000} C_DIS
LIN {X 54.858,Y -50.006,Z -204.663,A -90.000,B 90.000,C 0.000} C_DIS
LIN {X 54.664,Y -50.006,Z -206.086,A -90.000,B 90.000,C 0.000} C_DIS
LIN {X 54.411,Y -50.006,Z -207.499,A -90.000,B 90.000,C 0.000} C_DIS
LIN {X 54.099,Y -50.006,Z -208.901,A -90.000,B 90.000,C 0.000} C_DIS
LIN {X 53.729,Y -50.006,Z -210.288,A -90.000,B 90.000,C 0.000} C_DIS
LIN {X 53.300,Y -50.006,Z -211.658,A -90.000,B 90.000,C 0.000} C_DIS
LIN {X 52.818,Y -50.006,Z -213.786,A -90.000,B 90.000,C 0.000} C_DIS
LIN {X 52.286,Y -50.006,Z -215.902,A -90.000,B 90.000,C 0.000} C_DIS
LIN {X 51.704,Y -50.006,Z -218.004,A -90.000,B 90.000,C 0.000} C_DIS
LIN {X 51.072,Y -50.006,Z -220.093,A -90.000,B 90.000,C 0.000} C_DIS
LIN {X 50.391,Y -50.006,Z -222.166,A -90.000,B 90.000,C 0.000} C_DIS
LIN {X 49.662,Y -50.006,Z -224.222,A -90.000,B 90.000,C 0.000} C_DIS
LIN {X 48.894,Y -50.006,Z -225.918,A -90.000,B 90.000,C 0.000} C_DIS
LIN {X 48.071,Y -50.006,Z -227.588,A -90.000,B 90.000,C 0.000} C_DIS
LIN {X 47.193,Y -50.006,Z -229.230,A -90.000,B 90.000,C 0.000} C_DIS
LIN {X 46.262,Y -50.006,Z -230.842,A -90.000,B 90.000,C 0.000} C_DIS
LIN {X 45.278,Y -50.006,Z -232.422,A -90.000,B 90.000,C 0.000} C_DIS
LIN {X 44.060,Y -50.006,Z -233.779,A -90.000,B 90.000,C 0.000} C_DIS
LIN {X 42.804,Y -50.006,Z -235.101,A -90.000,B 90.000,C 0.000} C_DIS
LIN {X 41.511,Y -50.006,Z -236.386,A -90.000,B 90.000,C 0.000} C_DIS
LIN {X 40.182,Y -50.006,Z -237.634,A -90.000,B 90.000,C 0.000} C_DIS
LIN {X 38.818,Y -50.006,Z -238.844,A -90.000,B 90.000,C 0.000} C_DIS
LIN {X 37.684,Y -50.006,Z -239.531,A -90.000,B 90.000,C 0.000} C_DIS
LIN {X 36.530,Y -50.006,Z -240.184,A -90.000,B 90.000,C 0.000} C_DIS
LIN {X 35.358,Y -50.006,Z -240.804,A -90.000,B 90.000,C 0.000} C_DIS
LIN {X 34.168,Y -50.006,Z -241.389,A -90.000,B 90.000,C 0.000} C_DIS
LIN {X 33.463,Y -50.006,Z -241.742,A -90.000,B 90.000,C 0.000} C_DIS
LIN {X 32.731,Y -50.006,Z -242.035,A -90.000,B 90.000,C 0.000} C_DIS
LIN {X 31.977,Y -50.006,Z -242.267,A -90.000,B 90.000,C 0.000} C_DIS
LIN {X 31.207,Y -50.006,Z -242.436,A -90.000,B 90.000,C 0.000} C_DIS
LIN {X 30.425,Y -50.006,Z -242.540,A -90.000,B 90.000,C 0.000} C_DIS
LIN {X 29.637,Y -50.006,Z -242.579,A -90.000,B 90.000,C 0.000} C_DIS
LIN {X 28.849,Y -50.006,Z -242.553,A -90.000,B 90.000,C 0.000} C_DIS
LIN {X 26.127,Y -50.006,Z -241.978,A -90.000,B 90.000,C 0.000} C_DIS
LIN {X 23.398,Y -50.006,Z -241.438,A -90.000,B 90.000,C 0.000} C_DIS
LIN {X 22.620,Y -50.006,Z -241.230,A -90.000,B 90.000,C 0.000} C_DIS
LIN {X 21.863,Y -50.006,Z -240.957,A -90.000,B 90.000,C 0.000} C_DIS
LIN {X 21.131,Y -50.006,Z -240.620,A -90.000,B 90.000,C 0.000} C_DIS
LIN {X 20.431,Y -50.006,Z -240.224,A -90.000,B 90.000,C 0.000} C_DIS
LIN {X 19.766,Y -50.006,Z -239.769,A -90.000,B 90.000,C 0.000} C_DIS
LIN {X 19.143,Y -50.006,Z -239.260,A -90.000,B 90.000,C 0.000} C_DIS
LIN {X 18.564,Y -50.006,Z -238.700,A -90.000,B 90.000,C 0.000} C_DIS
LIN {X 18.035,Y -50.006,Z -238.094,A -90.000,B 90.000,C 0.000} C_DIS
LIN {X 17.559,Y -50.006,Z -237.444,A -90.000,B 90.000,C 0.000} C_DIS
LIN {X 17.139,Y -50.006,Z -236.757,A -90.000,B 90.000,C 0.000} C_DIS
LIN {X 16.779,Y -50.006,Z -236.037,A -90.000,B 90.000,C 0.000} C_DIS
LIN {X 16.482,Y -50.006,Z -235.289,A -90.000,B 90.000,C 0.000} C_DIS
LIN {X 16.155,Y -50.006,Z -233.612,A -90.000,B 90.000,C 0.000} C_DIS
LIN {X 15.868,Y -50.006,Z -231.928,A -90.000,B 90.000,C 0.000} C_DIS
LIN {X 15.621,Y -50.006,Z -230.238,A -90.000,B 90.000,C 0.000} C_DIS
LIN {X 15.413,Y -50.006,Z -228.542,A -90.000,B 90.000,C 0.000} C_DIS
LIN {X 15.470,Y -50.006,Z -227.695,A -90.000,B 90.000,C 0.000} C_DIS
LIN {X 15.550,Y -50.006,Z -226.850,A -90.000,B 90.000,C 0.000} C_DIS
LIN {X 15.653,Y -50.006,Z -226.008,A -90.000,B 90.000,C 0.000} C_DIS
LIN {X 8.426,Y -50.006,Z -145.055,A -90.000,B 90.000,C 0.000} C_DIS
LIN {X 7.552,Y -50.006,Z -145.106,A -90.000,B 90.000,C 0.000} C_DIS
LIN {X 6.677,Y -50.006,Z -145.092,A -90.000,B 90.000,C 0.000} C_DIS
LIN {X 5.805,Y -50.006,Z -145.014,A -90.000,B 90.000,C 0.000} C_DIS
LIN {X 4.941,Y -50.006,Z -144.873,A -90.000,B 90.000,C 0.000} C_DIS
LIN {X 4.090,Y -50.006,Z -144.668,A -90.000,B 90.000,C 0.000} C_DIS
LIN {X 3.256,Y -50.006,Z -144.402,A -90.000,B 90.000,C 0.000} C_DIS
LIN {X 2.444,Y -50.006,Z -144.075,A -90.000,B 90.000,C 0.000} C_DIS
LIN {X 1.658,Y -50.006,Z -143.690,A -90.000,B 90.000,C 0.000} C_DIS
LIN {X 0.903,Y -50.006,Z -143.247,A -90.000,B 90.000,C 0.000} C_DIS
LIN {X 0.182,Y -50.006,Z -142.751,A -90.000,B 90.000,C 0.000} C_DIS
LIN {X -0.545,Y -50.006,Z -142.261,A -90.000,B 90.000,C 0.000} C_DIS
LIN {X -1.241,Y -50.006,Z -141.729,A -90.000,B 90.000,C 0.000} C_DIS
LIN {X -1.905,Y -50.006,Z -141.157,A -90.000,B 90.000,C 0.000} C_DIS
LIN {X -2.534,Y -50.006,Z -140.547,A -90.000,B 90.000,C 0.000} C_DIS
LIN {X -3.126,Y -50.006,Z -139.900,A -90.000,B 90.000,C 0.000} C_DIS
LIN {X -3.679,Y -50.006,Z -139.220,A -90.000,B 90.000,C 0.000} C_DIS
LIN {X -4.193,Y -50.006,Z -138.268,A -90.000,B 90.000,C 0.000} C_DIS
LIN {X -4.648,Y -50.006,Z -137.286,A -90.000,B 90.000,C 0.000} C_DIS
LIN {X -5.043,Y -50.006,Z -136.278,A -90.000,B 90.000,C 0.000} C_DIS
LIN {X -5.374,Y -50.006,Z -135.248,A -90.000,B 90.000,C 0.000} C_DIS
LIN {X -5.642,Y -50.006,Z -134.199,A -90.000,B 90.000,C 0.000} C_DIS
LIN {X -5.845,Y -50.006,Z -133.136,A -90.000,B 90.000,C 0.000} C_DIS
LIN {X -5.963,Y -50.006,Z -132.356,A -90.000,B 90.000,C 0.000} C_DIS
LIN {X -6.017,Y -50.006,Z -131.569,A -90.000,B 90.000,C 0.000} C_DIS
LIN {X -6.005,Y -50.006,Z -130.781,A -90.000,B 90.000,C 0.000} C_DIS
LIN {X -5.928,Y -50.006,Z -129.996,A -90.000,B 90.000,C 0.000} C_DIS
LIN {X -5.786,Y -50.006,Z -129.220,A -90.000,B 90.000,C 0.000} C_DIS
LIN {X -5.580,Y -50.006,Z -128.459,A -90.000,B 90.000,C 0.000} C_DIS
LIN {X -5.313,Y -50.006,Z -127.717,A -90.000,B 90.000,C 0.000} C_DIS
LIN {X -4.906,Y -50.006,Z -126.866,A -90.000,B 90.000,C 0.000} C_DIS
LIN {X -4.449,Y -50.006,Z -126.041,A -90.000,B 90.000,C 0.000} C_DIS
LIN {X -3.943,Y -50.006,Z -125.245,A -90.000,B 90.000,C 0.000} C_DIS
LIN {X -3.391,Y -50.006,Z -124.480,A -90.000,B 90.000,C 0.000} C_DIS
LIN {X -2.794,Y -50.006,Z -123.750,A -90.000,B 90.000,C 0.000} C_DIS
LIN {X -2.389,Y -50.006,Z -123.140,A -90.000,B 90.000,C 0.000} C_DIS
LIN {X -1.944,Y -50.006,Z -122.558,A -90.000,B 90.000,C 0.000} C_DIS
LIN {X -1.461,Y -50.006,Z -122.008,A -90.000,B 90.000,C 0.000} C_DIS
LIN {X -0.941,Y -50.006,Z -121.492,A -90.000,B 90.000,C 0.000} C_DIS
LIN {X -0.387,Y -50.006,Z -121.013,A -90.000,B 90.000,C 0.000} C_DIS
LIN {X 0.198,Y -50.006,Z -120.572,A -90.000,B 90.000,C 0.000} C_DIS
LIN {X 1.131,Y -50.006,Z -119.898,A -90.000,B 90.000,C 0.000} C_DIS
LIN {X 2.101,Y -50.006,Z -119.278,A -90.000,B 90.000,C 0.000} C_DIS
LIN {X 3.104,Y -50.006,Z -118.713,A -90.000,B 90.000,C 0.000} C_DIS
LIN {X 4.138,Y -50.006,Z -118.206,A -90.000,B 90.000,C 0.000} C_DIS
LIN {X 5.198,Y -50.006,Z -117.757,A -90.000,B 90.000,C 0.000} C_DIS
LIN {X 6.282,Y -50.006,Z -117.369,A -90.000,B 90.000,C 0.000} C_DIS
LIN {X 7.386,Y -50.006,Z -117.042,A -90.000,B 90.000,C 0.000} C_DIS
LIN {X 8.506,Y -50.006,Z -116.778,A -90.000,B 90.000,C 0.000} C_DIS
LIN {X 9.640,Y -50.006,Z -116.578,A -90.000,B 90.000,C 0.000} C_DIS
LIN {X 10.783,Y -50.006,Z -116.441,A -90.000,B 90.000,C 0.000} C_DIS
LIN {X 11.685,Y -50.006,Z -116.315,A -90.000,B 90.000,C 0.000} C_DIS
LIN {X 12.594,Y -50.006,Z -116.252,A -90.000,B 90.000,C 0.000} C_DIS
LIN {X 13.505,Y -50.006,Z -116.251,A -90.000,B 90.000,C 0.000} C_DIS
LIN {X 14.414,Y -50.006,Z -116.312,A -90.000,B 90.000,C 0.000} C_DIS
LIN {X 15.317,Y -50.006,Z -116.435,A -90.000,B 90.000,C 0.000} C_DIS
LIN {X 16.209,Y -50.006,Z -116.620,A -90.000,B 90.000,C 0.000} C_DIS
LIN {X 17.086,Y -50.006,Z -116.865,A -90.000,B 90.000,C 0.000} C_DIS
LIN {X 17.888,Y -50.006,Z -117.050,A -90.000,B 90.000,C 0.000} C_DIS
LIN {X 18.678,Y -50.006,Z -117.278,A -90.000,B 90.000,C 0.000} C_DIS
LIN {X 19.454,Y -50.006,Z -117.550,A -90.000,B 90.000,C 0.000} C_DIS
LIN {X 20.214,Y -50.006,Z -117.864,A -90.000,B 90.000,C 0.000} C_DIS
LIN {X 20.956,Y -50.006,Z -118.220,A -90.000,B 90.000,C 0.000} C_DIS
LIN {X 21.677,Y -50.006,Z -118.616,A -90.000,B 90.000,C 0.000} C_DIS
LIN {X 22.465,Y -50.006,Z -119.243,A -90.000,B 90.000,C 0.000} C_DIS
LIN {X 23.205,Y -50.006,Z -119.927,A -90.000,B 90.000,C 0.000} C_DIS
LIN {X 23.893,Y -50.006,Z -120.663,A -90.000,B 90.000,C 0.000} C_DIS
LIN {X 24.525,Y -50.006,Z -121.448,A -90.000,B 90.000,C 0.000} C_DIS
LIN {X 25.097,Y -50.006,Z -122.277,A -90.000,B 90.000,C 0.000} C_DIS
LIN {X 25.607,Y -50.006,Z -123.146,A -90.000,B 90.000,C 0.000} C_DIS
LIN {X 26.051,Y -50.006,Z -124.050,A -90.000,B 90.000,C 0.000} C_DIS
LIN {X 26.428,Y -50.006,Z -124.984,A -90.000,B 90.000,C 0.000} C_DIS
LIN {X 26.735,Y -50.006,Z -125.944,A -90.000,B 90.000,C 0.000} C_DIS
LIN {X 26.970,Y -50.006,Z -126.923,A -90.000,B 90.000,C 0.000} C_DIS
LIN {X 27.133,Y -50.006,Z -127.917,A -90.000,B 90.000,C 0.000} C_DIS
LIN {X 27.222,Y -50.006,Z -128.921,A -90.000,B 90.000,C 0.000} C_DIS
LIN {X 27.237,Y -50.006,Z -129.928,A -90.000,B 90.000,C 0.000} C_DIS
LIN {X 27.178,Y -50.006,Z -130.934,A -90.000,B 90.000,C 0.000} C_DIS
LIN {X 27.045,Y -50.006,Z -131.933,A -90.000,B 90.000,C 0.000} C_DIS
LIN {X 26.839,Y -50.006,Z -132.919,A -90.000,B 90.000,C 0.000} C_DIS
LIN {X 26.561,Y -50.006,Z -133.887,A -90.000,B 90.000,C 0.000} C_DIS
LIN {X 26.212,Y -50.006,Z -134.832,A -90.000,B 90.000,C 0.000} C_DIS
LIN {X 25.795,Y -50.006,Z -135.749,A -90.000,B 90.000,C 0.000} C_DIS
LIN {X 25.190,Y -50.006,Z -136.692,A -90.000,B 90.000,C 0.000} C_DIS
LIN {X 24.542,Y -50.006,Z -137.604,A -90.000,B 90.000,C 0.000} C_DIS
LIN {X 23.851,Y -50.006,Z -138.485,A -90.000,B 90.000,C 0.000} C_DIS
LIN {X 23.119,Y -50.006,Z -139.333,A -90.000,B 90.000,C 0.000} C_DIS
LIN {X 22.347,Y -50.006,Z -140.144,A -90.000,B 90.000,C 0.000} C_DIS
LIN {X 21.538,Y -50.006,Z -140.918,A -90.000,B 90.000,C 0.000} C_DIS
LIN {X 20.693,Y -50.006,Z -141.653,A -90.000,B 90.000,C 0.000} C_DIS
LIN {X 19.704,Y -50.006,Z -142.219,A -90.000,B 90.000,C 0.000} C_DIS
LIN {X 18.687,Y -50.006,Z -142.733,A -90.000,B 90.000,C 0.000} C_DIS
LIN {X 17.645,Y -50.006,Z -143.195,A -90.000,B 90.000,C 0.000} C_DIS
LIN {X 16.580,Y -50.006,Z -143.602,A -90.000,B 90.000,C 0.000} C_DIS
LIN {X 15.497,Y -50.006,Z -143.954,A -90.000,B 90.000,C 0.000} C_DIS
LIN {X 14.396,Y -50.006,Z -144.250,A -90.000,B 90.000,C 0.000} C_DIS
LIN {X 13.428,Y -50.006,Z -144.537,A -90.000,B 90.000,C 0.000} C_DIS
LIN {X 12.444,Y -50.006,Z -144.764,A -90.000,B 90.000,C 0.000} C_DIS
LIN {X 11.448,Y -50.006,Z -144.930,A -90.000,B 90.000,C 0.000} C_DIS
LIN {X 10.444,Y -50.006,Z -145.034,A -90.000,B 90.000,C 0.000} C_DIS
LIN {X 9.435,Y -50.006,Z -145.076,A -90.000,B 90.000,C 0.000} C_DIS
LIN {X 8.426,Y -50.006,Z -145.055,A -90.000,B 90.000,C 0.000} C_DIS
LIN {X 9.435,Y -50.006,Z -145.075,A -90.000,B 90.000,C 0.000} C_DIS
LIN {X 10.444,Y -50.006,Z -145.034,A -90.000,B 90.000,C 0.000} C_DIS
LIN {X 11.448,Y -50.006,Z -144.930,A -90.000,B 90.000,C 0.000} C_DIS
LIN {X 12.444,Y -50.006,Z -144.764,A -90.000,B 90.000,C 0.000} C_DIS
LIN {X 13.428,Y -50.006,Z -144.537,A -90.000,B 90.000,C 0.000} C_DIS
LIN {X 14.396,Y -50.006,Z -144.250,A -90.000,B 90.000,C 0.000} C_DIS
LIN {X 15.497,Y -50.006,Z -143.954,A -90.000,B 90.000,C 0.000} C_DIS
LIN {X 16.580,Y -50.006,Z -143.602,A -90.000,B 90.000,C 0.000} C_DIS
LIN {X 17.645,Y -50.006,Z -143.195,A -90.000,B 90.000,C 0.000} C_DIS
LIN {X 18.687,Y -50.006,Z -142.733,A -90.000,B 90.000,C 0.000} C_DIS
LIN {X 19.704,Y -50.006,Z -142.219,A -90.000,B 90.000,C 0.000} C_DIS
LIN {X 20.693,Y -50.006,Z -141.653,A -90.000,B 90.000,C 0.000} C_DIS
LIN {X 21.538,Y -50.006,Z -140.918,A -90.000,B 90.000,C 0.000} C_DIS
LIN {X 22.347,Y -50.006,Z -140.144,A -90.000,B 90.000,C 0.000} C_DIS
LIN {X 23.119,Y -50.006,Z -139.333,A -90.000,B 90.000,C 0.000} C_DIS
LIN {X 23.851,Y -50.006,Z -138.485,A -90.000,B 90.000,C 0.000} C_DIS
LIN {X 24.542,Y -50.006,Z -137.604,A -90.000,B 90.000,C 0.000} C_DIS
LIN {X 25.191,Y -50.006,Z -136.692,A -90.000,B 90.000,C 0.000} C_DIS
LIN {X 25.795,Y -50.006,Z -135.749,A -90.000,B 90.000,C 0.000} C_DIS
LIN {X 26.199,Y -50.006,Z -134.863,A -90.000,B 90.000,C 0.000} C_DIS
LIN {X 26.540,Y -50.006,Z -133.950,A -90.000,B 90.000,C 0.000} C_DIS
LIN {X 26.814,Y -50.006,Z -133.016,A -90.000,B 90.000,C 0.000} C_DIS
LIN {X 27.022,Y -50.006,Z -132.064,A -90.000,B 90.000,C 0.000} C_DIS
LIN {X 27.161,Y -50.006,Z -131.100,A -90.000,B 90.000,C 0.000} C_DIS
LIN {X 27.231,Y -50.006,Z -130.129,A -90.000,B 90.000,C 0.000} C_DIS
LIN {X 27.232,Y -50.006,Z -129.155,A -90.000,B 90.000,C 0.000} C_DIS
LIN {X 27.163,Y -50.006,Z -128.183,A -90.000,B 90.000,C 0.000} C_DIS
LIN {X 27.026,Y -50.006,Z -127.219,A -90.000,B 90.000,C 0.000} C_DIS
LIN {X 81.303,Y -50.006,Z -75.171,A -90.000,B 90.000,C 0.000} C_DIS
LIN {X 80.578,Y -50.006,Z -74.623,A -90.000,B 90.000,C 0.000} C_DIS
LIN {X 79.895,Y -50.006,Z -74.022,A -90.000,B 90.000,C 0.000} C_DIS
LIN {X 79.260,Y -50.006,Z -73.372,A -90.000,B 90.000,C 0.000} C_DIS
LIN {X 78.675,Y -50.006,Z -72.676,A -90.000,B 90.000,C 0.000} C_DIS
LIN {X 78.143,Y -50.006,Z -71.938,A -90.000,B 90.000,C 0.000} C_DIS
LIN {X 77.669,Y -50.006,Z -71.162,A -90.000,B 90.000,C 0.000} C_DIS
LIN {X 77.253,Y -50.006,Z -70.353,A -90.000,B 90.000,C 0.000} C_DIS
LIN {X 76.900,Y -50.006,Z -69.516,A -90.000,B 90.000,C 0.000} C_DIS
LIN {X 76.610,Y -50.006,Z -68.654,A -90.000,B 90.000,C 0.000} C_DIS
LIN {X 76.368,Y -50.006,Z -67.632,A -90.000,B 90.000,C 0.000} C_DIS
LIN {X 76.195,Y -50.006,Z -66.597,A -90.000,B 90.000,C 0.000} C_DIS
LIN {X 76.092,Y -50.006,Z -65.552,A -90.000,B 90.000,C 0.000} C_DIS
LIN {X 76.060,Y -50.006,Z -64.502,A -90.000,B 90.000,C 0.000} C_DIS
LIN {X 76.099,Y -50.006,Z -63.453,A -90.000,B 90.000,C 0.000} C_DIS
LIN {X 76.208,Y -50.006,Z -62.409,A -90.000,B 90.000,C 0.000} C_DIS
LIN {X 76.388,Y -50.006,Z -61.374,A -90.000,B 90.000,C 0.000} C_DIS
LIN {X 76.637,Y -50.006,Z -60.354,A -90.000,B 90.000,C 0.000} C_DIS
LIN {X 76.954,Y -50.006,Z -59.353,A -90.000,B 90.000,C 0.000} C_DIS
LIN {X 77.338,Y -50.006,Z -58.376,A -90.000,B 90.000,C 0.000} C_DIS
LIN {X 77.788,Y -50.006,Z -57.427,A -90.000,B 90.000,C 0.000} C_DIS
LIN {X 78.529,Y -50.006,Z -56.283,A -90.000,B 90.000,C 0.000} C_DIS
LIN {X 79.315,Y -50.006,Z -55.169,A -90.000,B 90.000,C 0.000} C_DIS
LIN {X 80.143,Y -50.006,Z -54.086,A -90.000,B 90.000,C 0.000} C_DIS
LIN {X 81.013,Y -50.006,Z -53.037,A -90.000,B 90.000,C 0.000} C_DIS
LIN {X 81.923,Y -50.006,Z -52.023,A -90.000,B 90.000,C 0.000} C_DIS
LIN {X 82.873,Y -50.006,Z -51.045,A -90.000,B 90.000,C 0.000} C_DIS
LIN {X 83.860,Y -50.006,Z -50.105,A -90.000,B 90.000,C 0.000} C_DIS
LIN {X 84.883,Y -50.006,Z -49.204,A -90.000,B 90.000,C 0.000} C_DIS
LIN {X 88.147,Y -50.006,Z -46.405,A -90.000,B 90.000,C 0.000} C_DIS
LIN {X 91.388,Y -50.006,Z -43.579,A -90.000,B 90.000,C 0.000} C_DIS
LIN {X 92.200,Y -50.006,Z -42.751,A -90.000,B 90.000,C 0.000} C_DIS
LIN {X 93.052,Y -50.006,Z -41.964,A -90.000,B 90.000,C 0.000} C_DIS
LIN {X 93.942,Y -50.006,Z -41.219,A -90.000,B 90.000,C 0.000} C_DIS
LIN {X 94.867,Y -50.006,Z -40.520,A -90.000,B 90.000,C 0.000} C_DIS
LIN {X 95.826,Y -50.006,Z -39.867,A -90.000,B 90.000,C 0.000} C_DIS
LIN {X 96.816,Y -50.006,Z -39.261,A -90.000,B 90.000,C 0.000} C_DIS
LIN {X 97.834,Y -50.006,Z -38.706,A -90.000,B 90.000,C 0.000} C_DIS
LIN {X 98.581,Y -50.006,Z -38.339,A -90.000,B 90.000,C 0.000} C_DIS
LIN {X 99.353,Y -50.006,Z -38.028,A -90.000,B 90.000,C 0.000} C_DIS
LIN {X 100.145,Y -50.006,Z -37.776,A -90.000,B 90.000,C 0.000} C_DIS
LIN {X 100.955,Y -50.006,Z -37.584,A -90.000,B 90.000,C 0.000} C_DIS
LIN {X 101.776,Y -50.006,Z -37.453,A -90.000,B 90.000,C 0.000} C_DIS
LIN {X 102.606,Y -50.006,Z -37.383,A -90.000,B 90.000,C 0.000} C_DIS
LIN {X 103.438,Y -50.006,Z -37.375,A -90.000,B 90.000,C 0.000} C_DIS
LIN {X 104.268,Y -50.006,Z -37.429,A -90.000,B 90.000,C 0.000} C_DIS
LIN {X 105.092,Y -50.006,Z -37.545,A -90.000,B 90.000,C 0.000} C_DIS
LIN {X 105.905,Y -50.006,Z -37.721,A -90.000,B 90.000,C 0.000} C_DIS
LIN {X 106.702,Y -50.006,Z -37.959,A -90.000,B 90.000,C 0.000} C_DIS
LIN {X 107.527,Y -50.006,Z -38.267,A -90.000,B 90.000,C 0.000} C_DIS
LIN {X 108.325,Y -50.006,Z -38.641,A -90.000,B 90.000,C 0.000} C_DIS
LIN {X 109.089,Y -50.006,Z -39.079,A -90.000,B 90.000,C 0.000} C_DIS
LIN {X 109.815,Y -50.006,Z -39.578,A -90.000,B 90.000,C 0.000} C_DIS
LIN {X 110.498,Y -50.006,Z -40.135,A -90.000,B 90.000,C 0.000} C_DIS
LIN {X 111.133,Y -50.006,Z -40.745,A -90.000,B 90.000,C 0.000} C_DIS
LIN {X 111.716,Y -50.006,Z -41.405,A -90.000,B 90.000,C 0.000} C_DIS
LIN {X 112.244,Y -50.006,Z -42.111,A -90.000,B 90.000,C 0.000} C_DIS
LIN {X 112.712,Y -50.006,Z -42.857,A -90.000,B 90.000,C 0.000} C_DIS
LIN {X 113.117,Y -50.006,Z -43.639,A -90.000,B 90.000,C 0.000} C_DIS
LIN {X 113.458,Y -50.006,Z -44.452,A -90.000,B 90.000,C 0.000} C_DIS
LIN {X 113.731,Y -50.006,Z -45.289,A -90.000,B 90.000,C 0.000} C_DIS
LIN {X 113.917,Y -50.006,Z -46.191,A -90.000,B 90.000,C 0.000} C_DIS
LIN {X 114.053,Y -50.006,Z -47.102,A -90.000,B 90.000,C 0.000} C_DIS
LIN {X 114.138,Y -50.006,Z -48.018,A -90.000,B 90.000,C 0.000} C_DIS
LIN {X 114.173,Y -50.006,Z -48.939,A -90.000,B 90.000,C 0.000} C_DIS
LIN {X 114.157,Y -50.006,Z -49.859,A -90.000,B 90.000,C 0.000} C_DIS
LIN {X 114.091,Y -50.006,Z -50.778,A -90.000,B 90.000,C 0.000} C_DIS
LIN {X 113.974,Y -50.006,Z -51.691,A -90.000,B 90.000,C 0.000} C_DIS
LIN {X 113.849,Y -50.006,Z -53.237,A -90.000,B 90.000,C 0.000} C_DIS
LIN {X 113.659,Y -50.006,Z -54.776,A -90.000,B 90.000,C 0.000} C_DIS
LIN {X 113.404,Y -50.006,Z -56.306,A -90.000,B 90.000,C 0.000} C_DIS
LIN {X 113.085,Y -50.006,Z -57.824,A -90.000,B 90.000,C 0.000} C_DIS
LIN {X 112.703,Y -50.006,Z -59.327,A -90.000,B 90.000,C 0.000} C_DIS
LIN {X 112.257,Y -50.006,Z -60.812,A -90.000,B 90.000,C 0.000} C_DIS
LIN {X 111.750,Y -50.006,Z -62.277,A -90.000,B 90.000,C 0.000} C_DIS
LIN {X 111.181,Y -50.006,Z -63.720,A -90.000,B 90.000,C 0.000} C_DIS
LIN {X 110.552,Y -50.006,Z -65.138,A -90.000,B 90.000,C 0.000} C_DIS
LIN {X 109.863,Y -50.006,Z -66.527,A -90.000,B 90.000,C 0.000} C_DIS
LIN {X 109.117,Y -50.006,Z -67.887,A -90.000,B 90.000,C 0.000} C_DIS
LIN {X 108.511,Y -50.006,Z -68.907,A -90.000,B 90.000,C 0.000} C_DIS
LIN {X 107.855,Y -50.006,Z -69.895,A -90.000,B 90.000,C 0.000} C_DIS
LIN {X 107.151,Y -50.006,Z -70.850,A -90.000,B 90.000,C 0.000} C_DIS
LIN {X 106.400,Y -50.006,Z -71.768,A -90.000,B 90.000,C 0.000} C_DIS
LIN {X 105.604,Y -50.006,Z -72.648,A -90.000,B 90.000,C 0.000} C_DIS
LIN {X 104.766,Y -50.006,Z -73.487,A -90.000,B 90.000,C 0.000} C_DIS
LIN {X 103.887,Y -50.006,Z -74.283,A -90.000,B 90.000,C 0.000} C_DIS
LIN {X 102.969,Y -50.006,Z -75.035,A -90.000,B 90.000,C 0.000} C_DIS
LIN {X 102.139,Y -50.006,Z -75.688,A -90.000,B 90.000,C 0.000} C_DIS
LIN {X 101.270,Y -50.006,Z -76.287,A -90.000,B 90.000,C 0.000} C_DIS
LIN {X 100.365,Y -50.006,Z -76.830,A -90.000,B 90.000,C 0.000} C_DIS
LIN {X 99.427,Y -50.006,Z -77.315,A -90.000,B 90.000,C 0.000} C_DIS
LIN {X 98.460,Y -50.006,Z -77.740,A -90.000,B 90.000,C 0.000} C_DIS
LIN {X 97.469,Y -50.006,Z -78.103,A -90.000,B 90.000,C 0.000} C_DIS
LIN {X 96.457,Y -50.006,Z -78.402,A -90.000,B 90.000,C 0.000} C_DIS
LIN {X 95.427,Y -50.006,Z -78.637,A -90.000,B 90.000,C 0.000} C_DIS
LIN {X 94.385,Y -50.006,Z -78.807,A -90.000,B 90.000,C 0.000} C_DIS
LIN {X 93.335,Y -50.006,Z -78.910,A -90.000,B 90.000,C 0.000} C_DIS
LIN {X 92.280,Y -50.006,Z -78.947,A -90.000,B 90.000,C 0.000} C_DIS
LIN {X 91.224,Y -50.006,Z -78.917,A -90.000,B 90.000,C 0.000} C_DIS
LIN {X 90.173,Y -50.006,Z -78.821,A -90.000,B 90.000,C 0.000} C_DIS
LIN {X 89.130,Y -50.006,Z -78.658,A -90.000,B 90.000,C 0.000} C_DIS
LIN {X 89.025,Y -50.006,Z -78.632,A -90.000,B 90.000,C 0.000} C_DIS
LIN {X 88.389,Y -50.006,Z -78.531,A -90.000,B 90.000,C 0.000} C_DIS
LIN {X 87.760,Y -50.006,Z -78.389,A -90.000,B 90.000,C 0.000} C_DIS
LIN {X 87.143,Y -50.006,Z -78.205,A -90.000,B 90.000,C 0.000} C_DIS
LIN {X 86.539,Y -50.006,Z -77.981,A -90.000,B 90.000,C 0.000} C_DIS
LIN {X 85.951,Y -50.006,Z -77.718,A -90.000,B 90.000,C 0.000} C_DIS
LIN {X 85.136,Y -50.006,Z -77.448,A -90.000,B 90.000,C 0.000} C_DIS
LIN {X 84.342,Y -50.006,Z -77.122,A -90.000,B 90.000,C 0.000} C_DIS
LIN {X 83.573,Y -50.006,Z -76.740,A -90.000,B 90.000,C 0.000} C_DIS
LIN {X 82.833,Y -50.006,Z -76.304,A -90.000,B 90.000,C 0.000} C_DIS
LIN {X 82.126,Y -50.006,Z -75.817,A -90.000,B 90.000,C 0.000} C_DIS
LIN {X 81.455,Y -50.006,Z -75.282,A -90.000,B 90.000,C 0.000} C_DIS
LIN {X 81.303,Y -50.006,Z -75.171,A -90.000,B 90.000,C 0.000} C_DIS
LIN {X 81.303,Y -62.506,Z -75.171,A -90.000,B 90.000,C 0.000} C_DIS
LIN {X 81.303,Y -75.006,Z -75.171,A -90.000,B 90.000,C 0.000} C_DIS
LIN {X -144.015,Y -75.006,Z -242.561,A -90.000,B 90.000,C 0.000} C_DIS
LIN {X -144.015,Y -67.862,Z -242.561,A -90.000,B 90.000,C 0.000} C_DIS
LIN {X -144.015,Y -55.362,Z -242.561,A -90.000,B 90.000,C 0.000} C_DIS
LIN {X -144.015,Y -42.862,Z -242.561,A -90.000,B 90.000,C 0.000} C_DIS
LIN {X -96.000,Y -42.862,Z -242.561,A -90.000,B 90.000,C 0.000} C_DIS
LIN {X -93.751,Y -42.862,Z -241.015,A -90.000,B 90.000,C 0.000} C_DIS
LIN {X -91.473,Y -42.862,Z -239.510,A -90.000,B 90.000,C 0.000} C_DIS
LIN {X -89.168,Y -42.862,Z -238.048,A -90.000,B 90.000,C 0.000} C_DIS
LIN {X -86.836,Y -42.862,Z -236.630,A -90.000,B 90.000,C 0.000} C_DIS
LIN {X -85.455,Y -42.862,Z -235.819,A -90.000,B 90.000,C 0.000} C_DIS
LIN {X -84.072,Y -42.862,Z -235.012,A -90.000,B 90.000,C 0.000} C_DIS
LIN {X -144.015,Y -42.862,Z -235.012,A -90.000,B 90.000,C 0.000} C_DIS
LIN {X -144.015,Y -42.862,Z -227.464,A -90.000,B 90.000,C 0.000} C_DIS
LIN {X -70.542,Y -42.862,Z -227.464,A -90.000,B 90.000,C 0.000} C_DIS
LIN {X -66.886,Y -42.862,Z -225.527,A -90.000,B 90.000,C 0.000} C_DIS
LIN {X -63.213,Y -42.862,Z -223.623,A -90.000,B 90.000,C 0.000} C_DIS
LIN {X -59.523,Y -42.862,Z -221.752,A -90.000,B 90.000,C 0.000} C_DIS
LIN {X -55.816,Y -42.862,Z -219.915,A -90.000,B 90.000,C 0.000} C_DIS
LIN {X -144.015,Y -42.862,Z -219.915,A -90.000,B 90.000,C 0.000} C_DIS
LIN {X -144.015,Y -42.862,Z -212.366,A -90.000,B 90.000,C 0.000} C_DIS
LIN {X -39.907,Y -42.862,Z -212.366,A -90.000,B 90.000,C 0.000} C_DIS
LIN {X -36.540,Y -42.862,Z -210.734,A -90.000,B 90.000,C 0.000} C_DIS
LIN {X -33.193,Y -42.862,Z -209.063,A -90.000,B 90.000,C 0.000} C_DIS
LIN {X -31.013,Y -42.862,Z -208.082,A -90.000,B 90.000,C 0.000} C_DIS
LIN {X -28.859,Y -42.862,Z -207.047,A -90.000,B 90.000,C 0.000} C_DIS
LIN {X -26.731,Y -42.862,Z -205.959,A -90.000,B 90.000,C 0.000} C_DIS
LIN {X -24.631,Y -42.862,Z -204.817,A -90.000,B 90.000,C 0.000} C_DIS
LIN {X -144.015,Y -42.862,Z -204.817,A -90.000,B 90.000,C 0.000} C_DIS
LIN {X -144.015,Y -42.862,Z -197.269,A -90.000,B 90.000,C 0.000} C_DIS
LIN {X -12.600,Y -42.862,Z -197.269,A -90.000,B 90.000,C 0.000} C_DIS
LIN {X -10.671,Y -42.862,Z -195.854,A -90.000,B 90.000,C 0.000} C_DIS
LIN {X -8.778,Y -42.862,Z -194.391,A -90.000,B 90.000,C 0.000} C_DIS
LIN {X -6.923,Y -42.862,Z -192.880,A -90.000,B 90.000,C 0.000} C_DIS
LIN {X -5.107,Y -42.862,Z -191.322,A -90.000,B 90.000,C 0.000} C_DIS
LIN {X -3.330,Y -42.862,Z -189.720,A -90.000,B 90.000,C 0.000} C_DIS
LIN {X -144.015,Y -42.862,Z -189.720,A -90.000,B 90.000,C 0.000} C_DIS
LIN {X -144.015,Y -42.862,Z -182.171,A -90.000,B 90.000,C 0.000} C_DIS
LIN {X 3.942,Y -42.862,Z -182.171,A -90.000,B 90.000,C 0.000} C_DIS
LIN {X 5.656,Y -42.862,Z -180.239,A -90.000,B 90.000,C 0.000} C_DIS
LIN {X 7.403,Y -42.862,Z -178.337,A -90.000,B 90.000,C 0.000} C_DIS
LIN {X 9.182,Y -42.862,Z -176.464,A -90.000,B 90.000,C 0.000} C_DIS
LIN {X 10.992,Y -42.862,Z -174.622,A -90.000,B 90.000,C 0.000} C_DIS
LIN {X -144.015,Y -42.862,Z -174.622,A -90.000,B 90.000,C 0.000} C_DIS
LIN {X -144.015,Y -42.862,Z -167.073,A -90.000,B 90.000,C 0.000} C_DIS
LIN {X 18.766,Y -42.862,Z -167.073,A -90.000,B 90.000,C 0.000} C_DIS
LIN {X 19.644,Y -42.862,Z -166.054,A -90.000,B 90.000,C 0.000} C_DIS
LIN {X 20.491,Y -42.862,Z -165.009,A -90.000,B 90.000,C 0.000} C_DIS
LIN {X 21.308,Y -42.862,Z -163.940,A -90.000,B 90.000,C 0.000} C_DIS
LIN {X 22.092,Y -42.862,Z -162.848,A -90.000,B 90.000,C 0.000} C_DIS
LIN {X 22.845,Y -42.862,Z -161.733,A -90.000,B 90.000,C 0.000} C_DIS
LIN {X 23.611,Y -42.862,Z -160.640,A -90.000,B 90.000,C 0.000} C_DIS
LIN {X 24.345,Y -42.862,Z -159.525,A -90.000,B 90.000,C 0.000} C_DIS
LIN {X -144.015,Y -42.862,Z -159.525,A -90.000,B 90.000,C 0.000} C_DIS
LIN {X -144.015,Y -42.862,Z -151.976,A -90.000,B 90.000,C 0.000} C_DIS
LIN {X -19.012,Y -42.862,Z -151.976,A -90.000,B 90.000,C 0.000} C_DIS
LIN {X -20.513,Y -42.862,Z -150.984,A -90.000,B 90.000,C 0.000} C_DIS
LIN {X -21.977,Y -42.862,Z -149.938,A -90.000,B 90.000,C 0.000} C_DIS
LIN {X -23.403,Y -42.862,Z -148.841,A -90.000,B 90.000,C 0.000} C_DIS
LIN {X -24.788,Y -42.862,Z -147.693,A -90.000,B 90.000,C 0.000} C_DIS
LIN {X -26.132,Y -42.862,Z -146.496,A -90.000,B 90.000,C 0.000} C_DIS
LIN {X -27.431,Y -42.862,Z -145.252,A -90.000,B 90.000,C 0.000} C_DIS
LIN {X -27.801,Y -42.862,Z -144.842,A -90.000,B 90.000,C 0.000} C_DIS
LIN {X -28.165,Y -42.862,Z -144.427,A -90.000,B 90.000,C 0.000} C_DIS
LIN {X -144.015,Y -42.862,Z -144.427,A -90.000,B 90.000,C 0.000} C_DIS
LIN {X -144.015,Y -42.862,Z -136.878,A -90.000,B 90.000,C 0.000} C_DIS
LIN {X -33.365,Y -42.862,Z -136.878,A -90.000,B 90.000,C 0.000} C_DIS
LIN {X -33.998,Y -42.862,Z -135.649,A -90.000,B 90.000,C 0.000} C_DIS
LIN {X -34.590,Y -42.862,Z -134.400,A -90.000,B 90.000,C 0.000} C_DIS
LIN {X -35.140,Y -42.862,Z -133.132,A -90.000,B 90.000,C 0.000} C_DIS
LIN {X -35.647,Y -42.862,Z -131.847,A -90.000,B 90.000,C 0.000} C_DIS
LIN {X -36.111,Y -42.862,Z -130.545,A -90.000,B 90.000,C 0.000} C_DIS
LIN {X -36.426,Y -42.862,Z -129.944,A -90.000,B 90.000,C 0.000} C_DIS
LIN {X -36.713,Y -42.862,Z -129.329,A -90.000,B 90.000,C 0.000} C_DIS
LIN {X -144.015,Y -42.862,Z -129.329,A -90.000,B 90.000,C 0.000} C_DIS
LIN {X -144.015,Y -42.862,Z -121.781,A -90.000,B 90.000,C 0.000} C_DIS
LIN {X -39.403,Y -42.862,Z -121.781,A -90.000,B 90.000,C 0.000} C_DIS
LIN {X -39.756,Y -42.862,Z -120.738,A -90.000,B 90.000,C 0.000} C_DIS
LIN {X -40.077,Y -42.862,Z -119.684,A -90.000,B 90.000,C 0.000} C_DIS
LIN {X -40.107,Y -42.862,Z -119.526,A -90.000,B 90.000,C 0.000} C_DIS
LIN {X -40.158,Y -42.862,Z -119.350,A -90.000,B 90.000,C 0.000} C_DIS
LIN {X -40.623,Y -42.862,Z -117.132,A -90.000,B 90.000,C 0.000} C_DIS
LIN {X -41.123,Y -42.862,Z -114.921,A -90.000,B 90.000,C 0.000} C_DIS
LIN {X -41.194,Y -42.862,Z -114.232,A -90.000,B 90.000,C 0.000} C_DIS
LIN {X -144.015,Y -42.862,Z -114.232,A -90.000,B 90.000,C 0.000} C_DIS
